LIN {X 0,Y 112.614,Z 722.748,A -85,B 0,C 180,E1 -26395.902,E2 -26395.902} C_VEL
LIN {X 0,Y 117.98,Z 722.724,A -85,B 0,C 180,E1 -26402.419,E2 -26402.419} C_VEL
LIN {X 0,Y 125.127,Z 721.325,A -85,B 0,C 180,E1 -26408.157,E2 -26408.157} C_VEL
LIN {X 0,Y 133.921,Z 718.463,A -85,B 0,C 180,E1 -26413.016,E2 -26413.016} C_VEL
LIN {X 0,Y 141.325,Z 715.337,A -85,B 0,C 180,E1 -26416.142,E2 -26416.142} C_VEL
LIN {X 0,Y 149.284,Z 711.254,A -85,B 0,C 180,E1 -26418.871,E2 -26418.871} C_VEL
LIN {X 0,Y 158.633,Z 705.602,A -85,B 0,C 180,E1 -26421.472,E2 -26421.472} C_VEL
LIN {X 0,Y 168.139,Z 698.779,A -85,B 0,C 180,E1 -26423.572,E2 -26423.572} C_VEL
LIN {X 0,Y 177.498,Z 690.89,A -85,B 0,C 180,E1 -26425.242,E2 -26425.242} C_VEL
LIN {X 0,Y 187.18,Z 681.241,A -85,B 0,C 180,E1 -26426.63,E2 -26426.63} C_VEL
LIN {X 0,Y 190.089,Z 677.932,A -85,B 0,C 180,E1 -26427.016,E2 -26427.016} C_VEL
LIN {X 0,Y 190.338,Z 677.404,A -85,B 0,C 180,E1 -26427.586,E2 -26427.586} C_VEL
LIN {X 0,Y 181.04,Z 686.04,A -85,B 0,C 180,E1 -26429.692,E2 -26429.692} C_VEL
LIN {X 0,Y 172.667,Z 692.227,A -85,B 0,C 180,E1 -26431.786,E2 -26431.786} C_VEL
LIN {X 0,Y 168.26,Z 695.049,A -85,B 0,C 180,E1 -26432.741,E2 -26432.741} C_VEL
LIN {X 0,Y 156.692,Z 701.204,A -85,B 0,C 180,E1 -26434.37,E2 -26434.37} C_VEL
LIN {X 0,Y 150.109,Z 703.856,A -85,B 0,C 180,E1 -26435.619,E2 -26435.619} C_VEL
LIN {X 0,Y 147.136,Z 704.728,A -85,B 0,C 180,E1 -26436.515,E2 -26436.515} C_VEL
LIN {X 0,Y 139.812,Z 706.451,A -85,B 0,C 180,E1 -26439.399,E2 -26439.399} C_VEL
LIN {X 0,Y 132.422,Z 707.283,A -85,B 0,C 180,E1 -26442.801,E2 -26442.801} C_VEL
LIN {X 0,Y 124.975,Z 707.111,A -85,B 0,C 180,E1 -26447.002,E2 -26447.002} C_VEL
LIN {X 0,Y 120.601,Z 706.402,A -85,B 0,C 180,E1 -26449.933,E2 -26449.933} C_VEL
LIN {X 0,Y 116.605,Z 705.225,A -85,B 0,C 180,E1 -26453.078,E2 -26453.078} C_VEL
LIN {X 0,Y 112.62,Z 703.398,A -85,B 0,C 180,E1 -26456.804,E2 -26456.804} C_VEL
LIN {X 0,Y 108.337,Z 700.237,A -85,B 0,C 180,E1 -26461.86,E2 -26461.86} C_VEL
LIN {X 0,Y 104.736,Z 695.693,A -85,B 0,C 180,E1 -26467.714,E2 -26467.714} C_VEL
LIN {X 0,Y 102.439,Z 690.321,A -85,B 0,C 180,E1 -26473.505,E2 -26473.505} C_VEL
LIN {X 0,Y 101.184,Z 683.981,A -85,B 0,C 180,E1 -26479.266,E2 -26479.266} C_VEL
LIN {X 0,Y 100.922,Z 675.313,A -85,B 0,C 180,E1 -26485.69,E2 -26485.69} C_VEL
LIN {X 0,Y 101.574,Z 666.056,A -85,B 0,C 180,E1 -26491.262,E2 -26491.262} C_VEL
LIN {X 0,Y 102.776,Z 655.496,A -85,B 0,C 180,E1 -26496.342,E2 -26496.342} C_VEL
LIN {X 0,Y 104.173,Z 644.669,A -85,B 0,C 180,E1 -26500.495,E2 -26500.495} C_VEL
LIN {X 0,Y 105.616,Z 633.785,A -85,B 0,C 180,E1 -26503.761,E2 -26503.761} C_VEL
LIN {X 0,Y 107.07,Z 621.558,A -85,B 0,C 180,E1 -26506.565,E2 -26506.565} C_VEL
LIN {X 0,Y 108.307,Z 608.423,A -85,B 0,C 180,E1 -26508.73,E2 -26508.73} C_VEL
LIN {X 0,Y 109.201,Z 592.336,A -85,B 0,C 180,E1 -26510.542,E2 -26510.542} C_VEL
LIN {X 0,Y 101.07,Z 563.812,A -85,B 0,C 180,E1 -26514.537,E2 -26514.537} C_VEL
LIN {X 0,Y 100.847,Z 562.869,A -85,B 0,C 180,E1 -26515.21,E2 -26515.21} C_VEL
LIN {X 0,Y 100.671,Z 562.758,A -85,B 0,C 180,E1 -26520.747,E2 -26520.747} C_VEL
LIN {X 0,Y 100.789,Z 562.741,A -85,B 0,C 180,E1 -26525.269,E2 -26525.269} C_VEL
LIN {X 0,Y 100.817,Z 562.74,A -85,B 0,C 180,E1 -26529.602,E2 -26529.602} C_VEL
LIN {X 0,Y 101.107,Z 562.702,A -85,B 0,C 180,E1 -26536.699,E2 -26536.699} C_VEL
LIN {X 0,Y 101.245,Z 562.678,A -85,B 0,C 180,E1 -26542.02,E2 -26542.02} C_VEL
LIN {X 0,Y 101.869,Z 562.602,A -85,B 0,C 180,E1 -26550,E2 -26550} C_VEL
LIN {X 0,Y 101.245,Z 562.683,A -85,B 0,C 180,E1 -26557.98,E2 -26557.98} C_VEL
LIN {X 0,Y 101.104,Z 562.702,A -85,B 0,C 180,E1 -26563.294,E2 -26563.294} C_VEL
LIN {X 0,Y 100.819,Z 562.733,A -85,B 0,C 180,E1 -26570.398,E2 -26570.398} C_VEL
LIN {X 0,Y 100.777,Z 562.743,A -85,B 0,C 180,E1 -26574.958,E2 -26574.958} C_VEL
LIN {X 0,Y 100.708,Z 562.752,A -85,B 0,C 180,E1 -26583.127,E2 -26583.127} C_VEL
LIN {X 0,Y 100.695,Z 562.753,A -85,B 0,C 180,E1 -26589.846,E2 -26589.846} C_VEL
LIN {X 0,Y 100.689,Z 562.747,A -85,B 0,C 180,E1 -26595.732,E2 -26595.732} C_VEL
LIN {X 0,Y 100.662,Z 562.758,A -85,B 0,C 180,E1 -26601.069,E2 -26601.069} C_VEL
LIN {X 0,Y 100.701,Z 562.751,A -85,B 0,C 180,E1 -26606.874,E2 -26606.874} C_VEL
LIN {X 0,Y 100.786,Z 562.739,A -85,B 0,C 180,E1 -26615.265,E2 -26615.265} C_VEL
LIN {X 0,Y 100.821,Z 562.738,A -85,B 0,C 180,E1 -26619.6,E2 -26619.6} C_VEL
LIN {X 0,Y 101.188,Z 562.693,A -85,B 0,C 180,E1 -26627.972,E2 -26627.972} C_VEL
LIN {X 0,Y 101.267,Z 562.675,A -85,B 0,C 180,E1 -26632.02,E2 -26632.02} C_VEL
LIN {X 0,Y 101.867,Z 562.601,A -85,B 0,C 180,E1 -26639.999,E2 -26639.999} C_VEL
LIN {X 0,Y 101.263,Z 562.678,A -85,B 0,C 180,E1 -26647.977,E2 -26647.977} C_VEL
LIN {X 0,Y 101.122,Z 562.701,A -85,B 0,C 180,E1 -26653.349,E2 -26653.349} C_VEL
LIN {X 0,Y 100.813,Z 562.736,A -85,B 0,C 180,E1 -26660.398,E2 -26660.398} C_VEL
LIN {X 0,Y 100.772,Z 562.741,A -85,B 0,C 180,E1 -26664.958,E2 -26664.958} C_VEL
LIN {X 0,Y 100.689,Z 562.753,A -85,B 0,C 180,E1 -26673.115,E2 -26673.115} C_VEL
LIN {X 0,Y 100.638,Z 562.761,A -85,B 0,C 180,E1 -26679.81,E2 -26679.81} C_VEL
LIN {X 0,Y 100.674,Z 562.757,A -85,B 0,C 180,E1 -26685.726,E2 -26685.726} C_VEL
LIN {X 0,Y 101.408,Z 562.905,A -85,B 0,C 180,E1 -26694.618,E2 -26694.618} C_VEL
LIN {X 0,Y 101.774,Z 563.975,A -85,B 0,C 180,E1 -26695.205,E2 -26695.205} C_VEL
LIN {X 0,Y 103.632,Z 569.648,A -85,B 0,C 180,E1 -26696.132,E2 -26696.132} C_VEL
LIN {X 0,Y 103.272,Z 600.843,A -85,B 0,C 180,E1 -26699.875,E2 -26699.875} C_VEL
LIN {X 0,Y 104.824,Z 644.068,A -85,B 0,C 180,E1 -26705.293,E2 -26705.293} C_VEL
LIN {X 0,Y 105.422,Z 656.065,A -85,B 0,C 180,E1 -26707.461,E2 -26707.461} C_VEL
LIN {X 0,Y 104.651,Z 667.818,A -85,B 0,C 180,E1 -26710.38,E2 -26710.38} C_VEL
LIN {X 0,Y 103.741,Z 677.783,A -85,B 0,C 180,E1 -26713.635,E2 -26713.635} C_VEL
LIN {X 0,Y 102.893,Z 688.58,A -85,B 0,C 180,E1 -26718.176,E2 -26718.176} C_VEL
LIN {X 0,Y 102.772,Z 696.112,A -85,B 0,C 180,E1 -26722.139,E2 -26722.139} C_VEL
LIN {X 0,Y 103.173,Z 703.754,A -85,B 0,C 180,E1 -26727.071,E2 -26727.071} C_VEL
LIN {X 0,Y 104.291,Z 709.858,A -85,B 0,C 180,E1 -26731.931,E2 -26731.931} C_VEL
LIN {X 0,Y 103.97,Z 711.518,A -85,B 0,C 180,E1 -26733.876,E2 -26733.876} C_VEL
LIN {X 0,Y 102.447,Z 715.261,A -85,B 0,C 180,E1 -26739.875,E2 -26739.875} C_VEL
LIN {X 0,Y 102.309,Z 718.051,A -85,B 0,C 180,E1 -26745.948,E2 -26745.948} C_VEL
LIN {X 0,Y 102.995,Z 719.41,A -85,B 0,C 180,E1 -26749.948,E2 -26749.948} C_VEL
LIN {X 0,Y 106.397,Z 721.105,A -85,B 0,C 180,E1 -26757.54,E2 -26757.54} C_VEL
LIN {X 0,Y 112.126,Z 721.458,A -85,B 0,C 180,E1 -26764.34,E2 -26764.34} C_VEL
LIN {X 0,Y 119.679,Z 720.429,A -85,B 0,C 180,E1 -26770.236,E2 -26770.236} C_VEL
LIN {X 0,Y 128.829,Z 718.027,A -85,B 0,C 180,E1 -26775.167,E2 -26775.167} C_VEL
LIN {X 0,Y 136.51,Z 715.246,A -85,B 0,C 180,E1 -26778.287,E2 -26778.287} C_VEL
LIN {X 0,Y 144.725,Z 711.612,A -85,B 0,C 180,E1 -26780.983,E2 -26780.983} C_VEL
LIN {X 0,Y 154.641,Z 706.256,A -85,B 0,C 180,E1 -26783.606,E2 -26783.606} C_VEL
LIN {X 0,Y 164.038,Z 700.248,A -85,B 0,C 180,E1 -26785.56,E2 -26785.56} C_VEL
LIN {X 0,Y 173.549,Z 693.028,A -85,B 0,C 180,E1 -26787.168,E2 -26787.168} C_VEL
LIN {X 0,Y 176.452,Z 690.599,A -85,B 0,C 180,E1 -26787.574,E2 -26787.574} C_VEL
LIN {X 0,Y 177.168,Z 689.792,A -85,B 0,C 180,E1 -26788.056,E2 -26788.056} C_VEL
LIN {X 0,Y 168.844,Z 695.339,A -85,B 0,C 180,E1 -26790.035,E2 -26790.035} C_VEL
LIN {X 0,Y 159.095,Z 700.398,A -85,B 0,C 180,E1 -26792.651,E2 -26792.651} C_VEL
LIN {X 0,Y 150.849,Z 703.626,A -85,B 0,C 180,E1 -26795.21,E2 -26795.21} C_VEL
LIN {X 0,Y 147.136,Z 704.728,A -85,B 0,C 180,E1 -26796.515,E2 -26796.515} C_VEL
LIN {X 0,Y 142.536,Z 706.017,A -85,B 0,C 180,E1 -26797.902,E2 -26797.902} C_VEL
LIN {X 0,Y 133.959,Z 707.764,A -85,B 0,C 180,E1 -26799.843,E2 -26799.843} C_VEL
LIN {X 0,Y 125.513,Z 708.563,A -85,B 0,C 180,E1 -26802.069,E2 -26802.069} C_VEL
LIN {X 0,Y 121.226,Z 708.373,A -85,B 0,C 180,E1 -26803.933,E2 -26803.933} C_VEL
LIN {X 0,Y 115.029,Z 707.323,A -85,B 0,C 180,E1 -26807.833,E2 -26807.833} C_VEL
LIN {X 0,Y 108.972,Z 705.197,A -85,B 0,C 180,E1 -26812.59,E2 -26812.59} C_VEL
LIN {X 0,Y 103.625,Z 701.961,A -85,B 0,C 180,E1 -26818.058,E2 -26818.058} C_VEL
LIN {X 0,Y 98.769,Z 696.798,A -85,B 0,C 180,E1 -26825.028,E2 -26825.028} C_VEL
LIN {X 0,Y 95.833,Z 690.877,A -85,B 0,C 180,E1 -26831.636,E2 -26831.636} C_VEL
LIN {X 0,Y 94.242,Z 683.557,A -85,B 0,C 180,E1 -26838.48,E2 -26838.48} C_VEL
LIN {X 0,Y 93.898,Z 674.309,A -85,B 0,C 180,E1 -26845.612,E2 -26845.612} C_VEL
LIN {X 0,Y 94.554,Z 664.987,A -85,B 0,C 180,E1 -26851.354,E2 -26851.354} C_VEL
LIN {X 0,Y 95.779,Z 654.409,A -85,B 0,C 180,E1 -26856.6,E2 -26856.6} C_VEL
LIN {X 0,Y 97.327,Z 642.456,A -85,B 0,C 180,E1 -26861.22,E2 -26861.22} C_VEL
LIN {X 0,Y 98.9,Z 630.748,A -85,B 0,C 180,E1 -26864.716,E2 -26864.716} C_VEL
LIN {X 0,Y 100.413,Z 617.425,A -85,B 0,C 180,E1 -26867.672,E2 -26867.672} C_VEL
LIN {X 0,Y 101.564,Z 603.656,A -85,B 0,C 180,E1 -26869.76,E2 -26869.76} C_VEL
LIN {X 0,Y 102.182,Z 593.607,A -85,B 0,C 180,E1 -26870.905,E2 -26870.905} C_VEL
LIN {X 0,Y 93.914,Z 564.332,A -85,B 0,C 180,E1 -26875.334,E2 -26875.334} C_VEL
LIN {X 0,Y 93.803,Z 563.659,A -85,B 0,C 180,E1 -26876.216,E2 -26876.216} C_VEL
LIN {X 0,Y 93.672,Z 563.629,A -85,B 0,C 180,E1 -26884.206,E2 -26884.206} C_VEL
LIN {X 0,Y 93.694,Z 563.627,A -85,B 0,C 180,E1 -26887.974,E2 -26887.974} C_VEL
LIN {X 0,Y 94.027,Z 563.584,A -85,B 0,C 180,E1 -26896.339,E2 -26896.339} C_VEL
LIN {X 0,Y 94.178,Z 563.559,A -85,B 0,C 180,E1 -26901.417,E2 -26901.417} C_VEL
LIN {X 0,Y 94.794,Z 563.483,A -85,B 0,C 180,E1 -26910,E2 -26910} C_VEL
LIN {X 0,Y 94.178,Z 563.562,A -85,B 0,C 180,E1 -26918.584,E2 -26918.584} C_VEL
LIN {X 0,Y 94.024,Z 563.585,A -85,B 0,C 180,E1 -26923.654,E2 -26923.654} C_VEL
LIN {X 0,Y 93.696,Z 563.625,A -85,B 0,C 180,E1 -26932.027,E2 -26932.027} C_VEL
LIN {X 0,Y 93.624,Z 563.63,A -85,B 0,C 180,E1 -26936.769,E2 -26936.769} C_VEL
LIN {X 0,Y 93.614,Z 563.634,A -85,B 0,C 180,E1 -26944.326,E2 -26944.326} C_VEL
LIN {X 0,Y 93.578,Z 563.64,A -85,B 0,C 180,E1 -26952.525,E2 -26952.525} C_VEL
LIN {X 0,Y 93.567,Z 563.642,A -85,B 0,C 180,E1 -26958.686,E2 -26958.686} C_VEL
LIN {X 0,Y 93.602,Z 563.631,A -85,B 0,C 180,E1 -26965.681,E2 -26965.681} C_VEL
LIN {X 0,Y 93.67,Z 563.621,A -85,B 0,C 180,E1 -26974.203,E2 -26974.203} C_VEL
LIN {X 0,Y 93.696,Z 563.626,A -85,B 0,C 180,E1 -26977.971,E2 -26977.971} C_VEL
LIN {X 0,Y 94.091,Z 563.577,A -85,B 0,C 180,E1 -26987.05,E2 -26987.05} C_VEL
LIN {X 0,Y 94.2,Z 563.554,A -85,B 0,C 180,E1 -26991.417,E2 -26991.417} C_VEL
LIN {X 0,Y 94.793,Z 563.482,A -85,B 0,C 180,E1 -26999.998,E2 -26999.998} C_VEL
LIN {X 0,Y 94.196,Z 563.556,A -85,B 0,C 180,E1 -27008.58,E2 -27008.58} C_VEL
LIN {X 0,Y 94.04,Z 563.583,A -85,B 0,C 180,E1 -27013.706,E2 -27013.706} C_VEL
LIN {X 0,Y 93.691,Z 563.626,A -85,B 0,C 180,E1 -27022.027,E2 -27022.027} C_VEL
LIN {X 0,Y 93.62,Z 563.627,A -85,B 0,C 180,E1 -27026.769,E2 -27026.769} C_VEL
LIN {X 0,Y 93.585,Z 563.635,A -85,B 0,C 180,E1 -27034.304,E2 -27034.304} C_VEL
LIN {X 0,Y 93.539,Z 563.644,A -85,B 0,C 180,E1 -27042.546,E2 -27042.546} C_VEL
LIN {X 0,Y 93.7,Z 563.626,A -85,B 0,C 180,E1 -27048.593,E2 -27048.593} C_VEL
LIN {X 0,Y 94.204,Z 563.779,A -85,B 0,C 180,E1 -27053.835,E2 -27053.835} C_VEL
LIN {X 0,Y 94.503,Z 564.713,A -85,B 0,C 180,E1 -27054.45,E2 -27054.45} C_VEL
LIN {X 0,Y 96.606,Z 570.603,A -85,B 0,C 180,E1 -27055.497,E2 -27055.497} C_VEL
LIN {X 0,Y 96.273,Z 602.738,A -85,B 0,C 180,E1 -27059.653,E2 -27059.653} C_VEL
LIN {X 0,Y 97.713,Z 642.777,A -85,B 0,C 180,E1 -27065.061,E2 -27065.061} C_VEL
LIN {X 0,Y 98.343,Z 655.818,A -85,B 0,C 180,E1 -27067.627,E2 -27067.627} C_VEL
LIN {X 0,Y 97.577,Z 667.437,A -85,B 0,C 180,E1 -27070.778,E2 -27070.778} C_VEL
LIN {X 0,Y 96.645,Z 678.326,A -85,B 0,C 180,E1 -27074.716,E2 -27074.716} C_VEL
LIN {X 0,Y 96.023,Z 687.428,A -85,B 0,C 180,E1 -27078.923,E2 -27078.923} C_VEL
LIN {X 0,Y 96.001,Z 695.694,A -85,B 0,C 180,E1 -27083.695,E2 -27083.695} C_VEL
LIN {X 0,Y 96.682,Z 703.137,A -85,B 0,C 180,E1 -27088.958,E2 -27088.958} C_VEL
LIN {X 0,Y 97.48,Z 706.871,A -85,B 0,C 180,E1 -27092.066,E2 -27092.066} C_VEL
LIN {X 0,Y 97.411,Z 708.801,A -85,B 0,C 180,E1 -27094.137,E2 -27094.137} C_VEL
LIN {X 0,Y 95.833,Z 712.817,A -85,B 0,C 180,E1 -27100.564,E2 -27100.564} C_VEL
LIN {X 0,Y 95.848,Z 716,A -85,B 0,C 180,E1 -27107.6,E2 -27107.6} C_VEL
LIN {X 0,Y 98.145,Z 718.518,A -85,B 0,C 180,E1 -27115.444,E2 -27115.444} C_VEL
LIN {X 0,Y 103.091,Z 719.881,A -85,B 0,C 180,E1 -27123.05,E2 -27123.05} C_VEL
LIN {X 0,Y 110.231,Z 719.92,A -85,B 0,C 180,E1 -27129.61,E2 -27129.61} C_VEL
LIN {X 0,Y 119.01,Z 718.623,A -85,B 0,C 180,E1 -27135.123,E2 -27135.123} C_VEL
LIN {X 0,Y 129.174,Z 715.958,A -85,B 0,C 180,E1 -27139.612,E2 -27139.612} C_VEL
LIN {X 0,Y 140.368,Z 711.805,A -85,B 0,C 180,E1 -27143.233,E2 -27143.233} C_VEL
LIN {X 0,Y 149.67,Z 707.434,A -85,B 0,C 180,E1 -27145.594,E2 -27145.594} C_VEL
LIN {X 0,Y 158.536,Z 702.476,A -85,B 0,C 180,E1 -27147.38,E2 -27147.38} C_VEL
LIN {X 0,Y 162.831,Z 699.761,A -85,B 0,C 180,E1 -27148.12,E2 -27148.12} C_VEL
LIN {X 0,Y 162.66,Z 699.588,A -85,B 0,C 180,E1 -27148.771,E2 -27148.771} C_VEL
LIN {X 0,Y 156.372,Z 702.462,A -85,B 0,C 180,E1 -27150.372,E2 -27150.372} C_VEL
LIN {X 0,Y 150.137,Z 704.754,A -85,B 0,C 180,E1 -27152.09,E2 -27152.09} C_VEL
LIN {X 0,Y 142.887,Z 706.741,A -85,B 0,C 180,E1 -27154.429,E2 -27154.429} C_VEL
LIN {X 0,Y 132.822,Z 708.424,A -85,B 0,C 180,E1 -27158.261,E2 -27158.261} C_VEL
LIN {X 0,Y 125.562,Z 708.674,A -85,B 0,C 180,E1 -27161.593,E2 -27161.593} C_VEL
LIN {X 0,Y 121.226,Z 708.373,A -85,B 0,C 180,E1 -27163.933,E2 -27163.933} C_VEL
LIN {X 0,Y 117.065,Z 707.982,A -85,B 0,C 180,E1 -27165.936,E2 -27165.936} C_VEL
LIN {X 0,Y 109.219,Z 706.798,A -85,B 0,C 180,E1 -27168.95,E2 -27168.95} C_VEL
LIN {X 0,Y 101.808,Z 704.734,A -85,B 0,C 180,E1 -27172.341,E2 -27172.341} C_VEL
LIN {X 0,Y 98.458,Z 702.962,A -85,B 0,C 180,E1 -27174.932,E2 -27174.932} C_VEL
LIN {X 0,Y 92.966,Z 697.676,A -85,B 0,C 180,E1 -27182.168,E2 -27182.168} C_VEL
LIN {X 0,Y 89.528,Z 691.801,A -85,B 0,C 180,E1 -27189.034,E2 -27189.034} C_VEL
LIN {X 0,Y 87.61,Z 685.1,A -85,B 0,C 180,E1 -27195.719,E2 -27195.719} C_VEL
LIN {X 0,Y 86.875,Z 676.928,A -85,B 0,C 180,E1 -27202.6,E2 -27202.6} C_VEL
LIN {X 0,Y 87.298,Z 666.901,A -85,B 0,C 180,E1 -27209.546,E2 -27209.546} C_VEL
LIN {X 0,Y 88.446,Z 655.795,A -85,B 0,C 180,E1 -27215.655,E2 -27215.655} C_VEL
LIN {X 0,Y 89.807,Z 645.151,A -85,B 0,C 180,E1 -27220.215,E2 -27220.215} C_VEL
LIN {X 0,Y 91.519,Z 632.797,A -85,B 0,C 180,E1 -27224.321,E2 -27224.321} C_VEL
LIN {X 0,Y 93.099,Z 619.497,A -85,B 0,C 180,E1 -27227.559,E2 -27227.559} C_VEL
LIN {X 0,Y 94.334,Z 606.24,A -85,B 0,C 180,E1 -27229.802,E2 -27229.802} C_VEL
LIN {X 0,Y 95.01,Z 594.162,A -85,B 0,C 180,E1 -27231.319,E2 -27231.319} C_VEL
LIN {X 0,Y 86.895,Z 565.312,A -85,B 0,C 180,E1 -27236.044,E2 -27236.044} C_VEL
LIN {X 0,Y 86.672,Z 564.554,A -85,B 0,C 180,E1 -27236.99,E2 -27236.99} C_VEL
LIN {X 0,Y 86.588,Z 564.511,A -85,B 0,C 180,E1 -27243.234,E2 -27243.234} C_VEL
LIN {X 0,Y 86.647,Z 564.502,A -85,B 0,C 180,E1 -27251.069,E2 -27251.069} C_VEL
LIN {X 0,Y 86.934,Z 564.466,A -85,B 0,C 180,E1 -27255.965,E2 -27255.965} C_VEL
LIN {X 0,Y 87.088,Z 564.445,A -85,B 0,C 180,E1 -27260.712,E2 -27260.712} C_VEL
LIN {X 0,Y 87.721,Z 564.364,A -85,B 0,C 180,E1 -27270,E2 -27270} C_VEL
LIN {X 0,Y 87.087,Z 564.442,A -85,B 0,C 180,E1 -27279.288,E2 -27279.288} C_VEL
LIN {X 0,Y 86.934,Z 564.469,A -85,B 0,C 180,E1 -27284.036,E2 -27284.036} C_VEL
LIN {X 0,Y 86.648,Z 564.495,A -85,B 0,C 180,E1 -27288.931,E2 -27288.931} C_VEL
LIN {X 0,Y 86.587,Z 564.506,A -85,B 0,C 180,E1 -27296.764,E2 -27296.764} C_VEL
LIN {X 0,Y 86.538,Z 564.511,A -85,B 0,C 180,E1 -27305.692,E2 -27305.692} C_VEL
LIN {X 0,Y 86.513,Z 564.519,A -85,B 0,C 180,E1 -27313.017,E2 -27313.017} C_VEL
LIN {X 0,Y 86.483,Z 564.524,A -85,B 0,C 180,E1 -27319.448,E2 -27319.448} C_VEL
LIN {X 0,Y 86.547,Z 564.508,A -85,B 0,C 180,E1 -27325.357,E2 -27325.357} C_VEL
LIN {X 0,Y 86.585,Z 564.503,A -85,B 0,C 180,E1 -27333.232,E2 -27333.232} C_VEL
LIN {X 0,Y 86.665,Z 564.497,A -85,B 0,C 180,E1 -27341.07,E2 -27341.07} C_VEL
LIN {X 0,Y 86.969,Z 564.463,A -85,B 0,C 180,E1 -27345.968,E2 -27345.968} C_VEL
LIN {X 0,Y 87.108,Z 564.438,A -85,B 0,C 180,E1 -27350.712,E2 -27350.712} C_VEL
LIN {X 0,Y 87.72,Z 564.362,A -85,B 0,C 180,E1 -27359.998,E2 -27359.998} C_VEL
LIN {X 0,Y 87.105,Z 564.438,A -85,B 0,C 180,E1 -27369.285,E2 -27369.285} C_VEL
LIN {X 0,Y 86.949,Z 564.467,A -85,B 0,C 180,E1 -27374.086,E2 -27374.086} C_VEL
LIN {X 0,Y 86.585,Z 564.511,A -85,B 0,C 180,E1 -27383.942,E2 -27383.942} C_VEL
LIN {X 0,Y 86.473,Z 564.522,A -85,B 0,C 180,E1 -27389.184,E2 -27389.184} C_VEL
LIN {X 0,Y 86.503,Z 564.513,A -85,B 0,C 180,E1 -27395.665,E2 -27395.665} C_VEL
LIN {X 0,Y 86.488,Z 564.522,A -85,B 0,C 180,E1 -27403.002,E2 -27403.002} C_VEL
LIN {X 0,Y 87.038,Z 564.64,A -85,B 0,C 180,E1 -27412.959,E2 -27412.959} C_VEL
LIN {X 0,Y 87.289,Z 565.429,A -85,B 0,C 180,E1 -27413.621,E2 -27413.621} C_VEL
LIN {X 0,Y 89.59,Z 572.071,A -85,B 0,C 180,E1 -27414.937,E2 -27414.937} C_VEL
LIN {X 0,Y 89.226,Z 603.646,A -85,B 0,C 180,E1 -27419.364,E2 -27419.364} C_VEL
LIN {X 0,Y 90.54,Z 641.544,A -85,B 0,C 180,E1 -27424.881,E2 -27424.881} C_VEL
LIN {X 0,Y 91.204,Z 654.519,A -85,B 0,C 180,E1 -27427.618,E2 -27427.618} C_VEL
LIN {X 0,Y 90.703,Z 664.594,A -85,B 0,C 180,E1 -27430.517,E2 -27430.517} C_VEL
LIN {X 0,Y 89.956,Z 674.381,A -85,B 0,C 180,E1 -27434.131,E2 -27434.131} C_VEL
LIN {X 0,Y 89.213,Z 684.978,A -85,B 0,C 180,E1 -27439.216,E2 -27439.216} C_VEL
LIN {X 0,Y 89.28,Z 693.53,A -85,B 0,C 180,E1 -27444.353,E2 -27444.353} C_VEL
LIN {X 0,Y 90.089,Z 701.136,A -85,B 0,C 180,E1 -27450,E2 -27450} C_VEL
LIN {X 0,Y 90.894,Z 704.957,A -85,B 0,C 180,E1 -27453.324,E2 -27453.324} C_VEL
LIN {X 0,Y 90.876,Z 705.941,A -85,B 0,C 180,E1 -27454.435,E2 -27454.435} C_VEL
LIN {X 0,Y 89.349,Z 710.165,A -85,B 0,C 180,E1 -27461.34,E2 -27461.34} C_VEL
LIN {X 0,Y 89.552,Z 713.951,A -85,B 0,C 180,E1 -27469.655,E2 -27469.655} C_VEL
LIN {X 0,Y 92.001,Z 716.468,A -85,B 0,C 180,E1 -27477.279,E2 -27477.279} C_VEL
LIN {X 0,Y 97.349,Z 718.193,A -85,B 0,C 180,E1 -27485.277,E2 -27485.277} C_VEL
LIN {X 0,Y 104.936,Z 718.599,A -85,B 0,C 180,E1 -27492.045,E2 -27492.045} C_VEL
LIN {X 0,Y 114.15,Z 717.73,A -85,B 0,C 180,E1 -27497.629,E2 -27497.629} C_VEL
LIN {X 0,Y 124.712,Z 715.5,A -85,B 0,C 180,E1 -27502.086,E2 -27502.086} C_VEL
LIN {X 0,Y 136.237,Z 711.881,A -85,B 0,C 180,E1 -27505.625,E2 -27505.625} C_VEL
LIN {X 0,Y 146.692,Z 707.546,A -85,B 0,C 180,E1 -27508.09,E2 -27508.09} C_VEL
LIN {X 0,Y 148.457,Z 706.694,A -85,B 0,C 180,E1 -27508.441,E2 -27508.441} C_VEL
LIN {X 0,Y 150.011,Z 705.845,A -85,B 0,C 180,E1 -27508.98,E2 -27508.98} C_VEL
LIN {X 0,Y 143.67,Z 707.653,A -85,B 0,C 180,E1 -27510.715,E2 -27510.715} C_VEL
LIN {X 0,Y 137.561,Z 708.931,A -85,B 0,C 180,E1 -27512.626,E2 -27512.626} C_VEL
LIN {X 0,Y 131.584,Z 709.723,A -85,B 0,C 180,E1 -27514.706,E2 -27514.706} C_VEL
LIN {X 0,Y 125.816,Z 710.066,A -85,B 0,C 180,E1 -27516.984,E2 -27516.984} C_VEL
LIN {X 0,Y 119.956,Z 709.899,A -85,B 0,C 180,E1 -27519.616,E2 -27519.616} C_VEL
LIN {X 0,Y 115.046,Z 709.332,A -85,B 0,C 180,E1 -27522.216,E2 -27522.216} C_VEL
LIN {X 0,Y 108.524,Z 707.824,A -85,B 0,C 180,E1 -27526.258,E2 -27526.258} C_VEL
LIN {X 0,Y 101.345,Z 704.812,A -85,B 0,C 180,E1 -27532.029,E2 -27532.029} C_VEL
LIN {X 0,Y 98.458,Z 702.962,A -85,B 0,C 180,E1 -27534.932,E2 -27534.932} C_VEL
LIN {X 0,Y 95.363,Z 700.961,A -85,B 0,C 180,E1 -27537.644,E2 -27537.644} C_VEL
LIN {X 0,Y 89.282,Z 697.082,A -85,B 0,C 180,E1 -27541.863,E2 -27541.863} C_VEL
LIN {X 0,Y 83.909,Z 692.396,A -85,B 0,C 180,E1 -27546.473,E2 -27546.473} C_VEL
LIN {X 0,Y 82.054,Z 689.238,A -85,B 0,C 180,E1 -27549.707,E2 -27549.707} C_VEL
LIN {X 0,Y 80.213,Z 680.7,A -85,B 0,C 180,E1 -27558.037,E2 -27558.037} C_VEL
LIN {X 0,Y 79.889,Z 672.496,A -85,B 0,C 180,E1 -27564.702,E2 -27564.702} C_VEL
LIN {X 0,Y 80.59,Z 662.201,A -85,B 0,C 180,E1 -27571.552,E2 -27571.552} C_VEL
LIN {X 0,Y 81.9,Z 651.041,A -85,B 0,C 180,E1 -27577.443,E2 -27577.443} C_VEL
LIN {X 0,Y 83.508,Z 639.148,A -85,B 0,C 180,E1 -27582.323,E2 -27582.323} C_VEL
LIN {X 0,Y 85.191,Z 626.492,A -85,B 0,C 180,E1 -27586.21,E2 -27586.21} C_VEL
LIN {X 0,Y 86.581,Z 613.937,A -85,B 0,C 180,E1 -27588.995,E2 -27588.995} C_VEL
LIN {X 0,Y 88.035,Z 595.646,A -85,B 0,C 180,E1 -27591.64,E2 -27591.64} C_VEL
LIN {X 0,Y 79.802,Z 566.307,A -85,B 0,C 180,E1 -27596.794,E2 -27596.794} C_VEL
LIN {X 0,Y 79.61,Z 565.44,A -85,B 0,C 180,E1 -27597.831,E2 -27597.831} C_VEL
LIN {X 0,Y 79.529,Z 565.392,A -85,B 0,C 180,E1 -27603.779,E2 -27603.779} C_VEL
LIN {X 0,Y 79.515,Z 565.393,A -85,B 0,C 180,E1 -27609.297,E2 -27609.297} C_VEL
LIN {X 0,Y 79.828,Z 565.349,A -85,B 0,C 180,E1 -27615.574,E2 -27615.574} C_VEL
LIN {X 0,Y 79.971,Z 565.333,A -85,B 0,C 180,E1 -27619.877,E2 -27619.877} C_VEL
LIN {X 0,Y 80.648,Z 565.245,A -85,B 0,C 180,E1 -27630,E2 -27630} C_VEL
LIN {X 0,Y 79.97,Z 565.327,A -85,B 0,C 180,E1 -27640.123,E2 -27640.123} C_VEL
LIN {X 0,Y 79.747,Z 565.364,A -85,B 0,C 180,E1 -27645.33,E2 -27645.33} C_VEL
LIN {X 0,Y 79.516,Z 565.387,A -85,B 0,C 180,E1 -27650.704,E2 -27650.704} C_VEL
LIN {X 0,Y 79.485,Z 565.387,A -85,B 0,C 180,E1 -27657.844,E2 -27657.844} C_VEL
LIN {X 0,Y 79.395,Z 565.408,A -85,B 0,C 180,E1 -27662.08,E2 -27662.08} C_VEL
LIN {X 0,Y 79.395,Z 565.4,A -85,B 0,C 180,E1 -27668.289,E2 -27668.289} C_VEL
LIN {X 0,Y 79.419,Z 565.397,A -85,B 0,C 180,E1 -27675.067,E2 -27675.067} C_VEL
LIN {X 0,Y 79.401,Z 565.403,A -85,B 0,C 180,E1 -27682.807,E2 -27682.807} C_VEL
LIN {X 0,Y 79.387,Z 565.407,A -85,B 0,C 180,E1 -27687.913,E2 -27687.913} C_VEL
LIN {X 0,Y 79.526,Z 565.382,A -85,B 0,C 180,E1 -27693.775,E2 -27693.775} C_VEL
LIN {X 0,Y 79.524,Z 565.391,A -85,B 0,C 180,E1 -27699.296,E2 -27699.296} C_VEL
LIN {X 0,Y 79.842,Z 565.351,A -85,B 0,C 180,E1 -27705.523,E2 -27705.523} C_VEL
LIN {X 0,Y 79.993,Z 565.327,A -85,B 0,C 180,E1 -27709.878,E2 -27709.878} C_VEL
LIN {X 0,Y 80.648,Z 565.243,A -85,B 0,C 180,E1 -27719.998,E2 -27719.998} C_VEL
LIN {X 0,Y 79.99,Z 565.325,A -85,B 0,C 180,E1 -27730.119,E2 -27730.119} C_VEL
LIN {X 0,Y 79.761,Z 565.36,A -85,B 0,C 180,E1 -27735.326,E2 -27735.326} C_VEL
LIN {X 0,Y 79.511,Z 565.39,A -85,B 0,C 180,E1 -27740.703,E2 -27740.703} C_VEL
LIN {X 0,Y 79.48,Z 565.389,A -85,B 0,C 180,E1 -27747.842,E2 -27747.842} C_VEL
LIN {X 0,Y 79.375,Z 565.41,A -85,B 0,C 180,E1 -27752.088,E2 -27752.088} C_VEL
LIN {X 0,Y 79.364,Z 565.408,A -85,B 0,C 180,E1 -27758.305,E2 -27758.305} C_VEL
LIN {X 0,Y 79.442,Z 565.403,A -85,B 0,C 180,E1 -27765.049,E2 -27765.049} C_VEL
LIN {X 0,Y 79.912,Z 565.6,A -85,B 0,C 180,E1 -27772.213,E2 -27772.213} C_VEL
LIN {X 0,Y 80.171,Z 566.484,A -85,B 0,C 180,E1 -27772.859,E2 -27772.859} C_VEL
LIN {X 0,Y 82.536,Z 573.093,A -85,B 0,C 180,E1 -27774.248,E2 -27774.248} C_VEL
LIN {X 0,Y 82.268,Z 609.726,A -85,B 0,C 180,E1 -27779.875,E2 -27779.875} C_VEL
LIN {X 0,Y 83.447,Z 640.405,A -85,B 0,C 180,E1 -27784.763,E2 -27784.763} C_VEL
LIN {X 0,Y 84.032,Z 652.558,A -85,B 0,C 180,E1 -27787.516,E2 -27787.516} C_VEL
LIN {X 0,Y 83.971,Z 659.247,A -85,B 0,C 180,E1 -27789.464,E2 -27789.464} C_VEL
LIN {X 0,Y 83.298,Z 670.161,A -85,B 0,C 180,E1 -27793.456,E2 -27793.456} C_VEL
LIN {X 0,Y 82.526,Z 680.316,A -85,B 0,C 180,E1 -27798.331,E2 -27798.331} C_VEL
LIN {X 0,Y 82.516,Z 689.541,A -85,B 0,C 180,E1 -27803.888,E2 -27803.888} C_VEL
LIN {X 0,Y 83.287,Z 697.673,A -85,B 0,C 180,E1 -27810,E2 -27810} C_VEL
LIN {X 0,Y 84.42,Z 702.905,A -85,B 0,C 180,E1 -27814.775,E2 -27814.775} C_VEL
LIN {X 0,Y 82.914,Z 707.425,A -85,B 0,C 180,E1 -27822.234,E2 -27822.234} C_VEL
LIN {X 0,Y 83.02,Z 710.914,A -85,B 0,C 180,E1 -27829.792,E2 -27829.792} C_VEL
LIN {X 0,Y 85.997,Z 714.314,A -85,B 0,C 180,E1 -27839.362,E2 -27839.362} C_VEL
LIN {X 0,Y 91.822,Z 716.359,A -85,B 0,C 180,E1 -27847.756,E2 -27847.756} C_VEL
LIN {X 0,Y 99.865,Z 717.171,A -85,B 0,C 180,E1 -27854.727,E2 -27854.727} C_VEL
LIN {X 0,Y 109.535,Z 716.682,A -85,B 0,C 180,E1 -27860.347,E2 -27860.347} C_VEL
LIN {X 0,Y 120.505,Z 714.906,A -85,B 0,C 180,E1 -27864.733,E2 -27864.733} C_VEL
LIN {X 0,Y 132.363,Z 711.807,A -85,B 0,C 180,E1 -27868.159,E2 -27868.159} C_VEL
LIN {X 0,Y 135.122,Z 710.886,A -85,B 0,C 180,E1 -27868.813,E2 -27868.813} C_VEL
LIN {X 0,Y 136.15,Z 710.367,A -85,B 0,C 180,E1 -27869.503,E2 -27869.503} C_VEL
LIN {X 0,Y 124.78,Z 711.419,A -85,B 0,C 180,E1 -27873.22,E2 -27873.22} C_VEL
LIN {X 0,Y 115.71,Z 711.047,A -85,B 0,C 180,E1 -27876.892,E2 -27876.892} C_VEL
LIN {X 0,Y 107.749,Z 709.787,A -85,B 0,C 180,E1 -27880.967,E2 -27880.967} C_VEL
LIN {X 0,Y 102.104,Z 708.1,A -85,B 0,C 180,E1 -27884.497,E2 -27884.497} C_VEL
LIN {X 0,Y 95.808,Z 705.236,A -85,B 0,C 180,E1 -27889.434,E2 -27889.434} C_VEL
LIN {X 0,Y 89.905,Z 701.096,A -85,B 0,C 180,E1 -27895.518,E2 -27895.518} C_VEL
LIN {X 0,Y 85.562,Z 696.165,A -85,B 0,C 180,E1 -27901.878,E2 -27901.878} C_VEL
LIN {X 0,Y 82.054,Z 689.238,A -85,B 0,C 180,E1 -27909.707,E2 -27909.707} C_VEL
LIN {X 0,Y 80.513,Z 685.919,A -85,B 0,C 180,E1 -27912.939,E2 -27912.939} C_VEL
LIN {X 0,Y 76.802,Z 679.791,A -85,B 0,C 180,E1 -27917.907,E2 -27917.907} C_VEL
LIN {X 0,Y 73.624,Z 672.989,A -85,B 0,C 180,E1 -27922.954,E2 -27922.954} C_VEL
LIN {X 0,Y 73.02,Z 668.647,A -85,B 0,C 180,E1 -27926.142,E2 -27926.142} C_VEL
LIN {X 0,Y 73.795,Z 658.917,A -85,B 0,C 180,E1 -27932.659,E2 -27932.659} C_VEL
LIN {X 0,Y 75.116,Z 648.27,A -85,B 0,C 180,E1 -27938.307,E2 -27938.307} C_VEL
LIN {X 0,Y 76.825,Z 635.781,A -85,B 0,C 180,E1 -27943.417,E2 -27943.417} C_VEL
LIN {X 0,Y 78.468,Z 623.339,A -85,B 0,C 180,E1 -27947.168,E2 -27947.168} C_VEL
LIN {X 0,Y 79.828,Z 610.28,A -85,B 0,C 180,E1 -27949.967,E2 -27949.967} C_VEL
LIN {X 0,Y 80.842,Z 596.222,A -85,B 0,C 180,E1 -27952.092,E2 -27952.092} C_VEL
LIN {X 0,Y 72.7,Z 567.049,A -85,B 0,C 180,E1 -27957.759,E2 -27957.759} C_VEL
LIN {X 0,Y 72.495,Z 566.324,A -85,B 0,C 180,E1 -27958.841,E2 -27958.841} C_VEL
LIN {X 0,Y 72.396,Z 566.277,A -85,B 0,C 180,E1 -27967.152,E2 -27967.152} C_VEL
LIN {X 0,Y 72.724,Z 566.233,A -85,B 0,C 180,E1 -27975.111,E2 -27975.111} C_VEL
LIN {X 0,Y 72.862,Z 566.221,A -85,B 0,C 180,E1 -27978.878,E2 -27978.878} C_VEL
LIN {X 0,Y 73.574,Z 566.126,A -85,B 0,C 180,E1 -27990,E2 -27990} C_VEL
LIN {X 0,Y 72.861,Z 566.213,A -85,B 0,C 180,E1 -28001.123,E2 -28001.123} C_VEL
LIN {X 0,Y 72.577,Z 566.254,A -85,B 0,C 180,E1 -28006.888,E2 -28006.888} C_VEL
LIN {X 0,Y 72.397,Z 566.279,A -85,B 0,C 180,E1 -28012.849,E2 -28012.849} C_VEL
LIN {X 0,Y 72.379,Z 566.274,A -85,B 0,C 180,E1 -28019.081,E2 -28019.081} C_VEL
LIN {X 0,Y 72.315,Z 566.282,A -85,B 0,C 180,E1 -28025.669,E2 -28025.669} C_VEL
LIN {X 0,Y 72.273,Z 566.293,A -85,B 0,C 180,E1 -28032.898,E2 -28032.898} C_VEL
LIN {X 0,Y 72.309,Z 566.29,A -85,B 0,C 180,E1 -28041.036,E2 -28041.036} C_VEL
LIN {X 0,Y 72.305,Z 566.281,A -85,B 0,C 180,E1 -28044.322,E2 -28044.322} C_VEL
LIN {X 0,Y 72.393,Z 566.278,A -85,B 0,C 180,E1 -28050.959,E2 -28050.959} C_VEL
LIN {X 0,Y 72.4,Z 566.279,A -85,B 0,C 180,E1 -28057.15,E2 -28057.15} C_VEL
LIN {X 0,Y 72.757,Z 566.231,A -85,B 0,C 180,E1 -28065.002,E2 -28065.002} C_VEL
LIN {X 0,Y 72.88,Z 566.217,A -85,B 0,C 180,E1 -28068.878,E2 -28068.878} C_VEL
LIN {X 0,Y 73.575,Z 566.124,A -85,B 0,C 180,E1 -28079.998,E2 -28079.998} C_VEL
LIN {X 0,Y 72.878,Z 566.214,A -85,B 0,C 180,E1 -28091.118,E2 -28091.118} C_VEL
LIN {X 0,Y 72.581,Z 566.249,A -85,B 0,C 180,E1 -28096.885,E2 -28096.885} C_VEL
LIN {X 0,Y 72.392,Z 566.28,A -85,B 0,C 180,E1 -28102.849,E2 -28102.849} C_VEL
LIN {X 0,Y 72.375,Z 566.277,A -85,B 0,C 180,E1 -28109.081,E2 -28109.081} C_VEL
LIN {X 0,Y 72.292,Z 566.283,A -85,B 0,C 180,E1 -28115.681,E2 -28115.681} C_VEL
LIN {X 0,Y 72.276,Z 566.292,A -85,B 0,C 180,E1 -28122.893,E2 -28122.893} C_VEL
LIN {X 0,Y 72.747,Z 566.465,A -85,B 0,C 180,E1 -28131.199,E2 -28131.199} C_VEL
LIN {X 0,Y 73.112,Z 567.625,A -85,B 0,C 180,E1 -28132.032,E2 -28132.032} C_VEL
LIN {X 0,Y 75.398,Z 574.035,A -85,B 0,C 180,E1 -28133.498,E2 -28133.498} C_VEL
LIN {X 0,Y 75.415,Z 620.491,A -85,B 0,C 180,E1 -28141.306,E2 -28141.306} C_VEL
LIN {X 0,Y 76.364,Z 640.892,A -85,B 0,C 180,E1 -28144.968,E2 -28144.968} C_VEL
LIN {X 0,Y 77.067,Z 654.644,A -85,B 0,C 180,E1 -28148.607,E2 -28148.607} C_VEL
LIN {X 0,Y 76.567,Z 665.625,A -85,B 0,C 180,E1 -28152.644,E2 -28152.644} C_VEL
LIN {X 0,Y 75.921,Z 675.277,A -85,B 0,C 180,E1 -28157.299,E2 -28157.299} C_VEL
LIN {X 0,Y 75.777,Z 685.167,A -85,B 0,C 180,E1 -28163.342,E2 -28163.342} C_VEL
LIN {X 0,Y 76.503,Z 693.909,A -85,B 0,C 180,E1 -28170,E2 -28170} C_VEL
LIN {X 0,Y 77.748,Z 699.588,A -85,B 0,C 180,E1 -28175.186,E2 -28175.186} C_VEL
LIN {X 0,Y 77.773,Z 700.511,A -85,B 0,C 180,E1 -28176.282,E2 -28176.282} C_VEL
LIN {X 0,Y 76.443,Z 705.895,A -85,B 0,C 180,E1 -28186.01,E2 -28186.01} C_VEL
LIN {X 0,Y 78.093,Z 710.324,A -85,B 0,C 180,E1 -28196.741,E2 -28196.741} C_VEL
LIN {X 0,Y 83.023,Z 713.359,A -85,B 0,C 180,E1 -28206.337,E2 -28206.337} C_VEL
LIN {X 0,Y 90.542,Z 715.177,A -85,B 0,C 180,E1 -28214.313,E2 -28214.313} C_VEL
LIN {X 0,Y 99.952,Z 715.694,A -85,B 0,C 180,E1 -28220.663,E2 -28220.663} C_VEL
LIN {X 0,Y 110.758,Z 714.997,A -85,B 0,C 180,E1 -28225.575,E2 -28225.575} C_VEL
LIN {X 0,Y 122.59,Z 713.053,A -85,B 0,C 180,E1 -28229.307,E2 -28229.307} C_VEL
LIN {X 0,Y 121.225,Z 712.804,A -85,B 0,C 180,E1 -28230.412,E2 -28230.412} C_VEL
LIN {X 0,Y 111.092,Z 712.101,A -85,B 0,C 180,E1 -28234.225,E2 -28234.225} C_VEL
LIN {X 0,Y 106.023,Z 711.257,A -85,B 0,C 180,E1 -28236.565,E2 -28236.565} C_VEL
LIN {X 0,Y 95.82,Z 708.17,A -85,B 0,C 180,E1 -28242.453,E2 -28242.453} C_VEL
LIN {X 0,Y 88.205,Z 704.239,A -85,B 0,C 180,E1 -28248.512,E2 -28248.512} C_VEL
LIN {X 0,Y 82.231,Z 699.411,A -85,B 0,C 180,E1 -28255.099,E2 -28255.099} C_VEL
LIN {X 0,Y 77.413,Z 693.012,A -85,B 0,C 180,E1 -28263.012,E2 -28263.012} C_VEL
LIN {X 0,Y 74.558,Z 685.892,A -85,B 0,C 180,E1 -28270.869,E2 -28270.869} C_VEL
LIN {X 0,Y 73.18,Z 678.338,A -85,B 0,C 180,E1 -28278.189,E2 -28278.189} C_VEL
LIN {X 0,Y 73.02,Z 668.647,A -85,B 0,C 180,E1 -28286.142,E2 -28286.142} C_VEL
LIN {X 0,Y 72.607,Z 664.26,A -85,B 0,C 180,E1 -28289.149,E2 -28289.149} C_VEL
LIN {X 0,Y 70.514,Z 656.427,A -85,B 0,C 180,E1 -28293.655,E2 -28293.655} C_VEL
LIN {X 0,Y 68.656,Z 648.054,A -85,B 0,C 180,E1 -28297.937,E2 -28297.937} C_VEL
LIN {X 0,Y 68.69,Z 642.762,A -85,B 0,C 180,E1 -28300.415,E2 -28300.415} C_VEL
LIN {X 0,Y 70.285,Z 631.381,A -85,B 0,C 180,E1 -28304.911,E2 -28304.911} C_VEL
LIN {X 0,Y 72.007,Z 617.616,A -85,B 0,C 180,E1 -28308.805,E2 -28308.805} C_VEL
LIN {X 0,Y 73.459,Z 601.642,A -85,B 0,C 180,E1 -28311.747,E2 -28311.747} C_VEL
LIN {X 0,Y 73.666,Z 596.873,A -85,B 0,C 180,E1 -28312.521,E2 -28312.521} C_VEL
LIN {X 0,Y 65.717,Z 568.366,A -85,B 0,C 180,E1 -28318.589,E2 -28318.589} C_VEL
LIN {X 0,Y 65.452,Z 567.294,A -85,B 0,C 180,E1 -28319.63,E2 -28319.63} C_VEL
LIN {X 0,Y 65.383,Z 567.149,A -85,B 0,C 180,E1 -28331.189,E2 -28331.189} C_VEL
LIN {X 0,Y 65.758,Z 567.107,A -85,B 0,C 180,E1 -28337.658,E2 -28337.658} C_VEL
LIN {X 0,Y 66.497,Z 567.007,A -85,B 0,C 180,E1 -28350,E2 -28350} C_VEL
LIN {X 0,Y 65.758,Z 567.101,A -85,B 0,C 180,E1 -28362.343,E2 -28362.343} C_VEL
LIN {X 0,Y 65.382,Z 567.143,A -85,B 0,C 180,E1 -28368.813,E2 -28368.813} C_VEL
LIN {X 0,Y 65.249,Z 567.167,A -85,B 0,C 180,E1 -28375.521,E2 -28375.521} C_VEL
LIN {X 0,Y 65.206,Z 567.175,A -85,B 0,C 180,E1 -28382.609,E2 -28382.609} C_VEL
LIN {X 0,Y 65.208,Z 567.175,A -85,B 0,C 180,E1 -28391.02,E2 -28391.02} C_VEL
LIN {X 0,Y 65.22,Z 567.173,A -85,B 0,C 180,E1 -28399.715,E2 -28399.715} C_VEL
LIN {X 0,Y 65.256,Z 567.169,A -85,B 0,C 180,E1 -28409.494,E2 -28409.494} C_VEL
LIN {X 0,Y 65.249,Z 567.161,A -85,B 0,C 180,E1 -28414.477,E2 -28414.477} C_VEL
LIN {X 0,Y 65.652,Z 567.114,A -85,B 0,C 180,E1 -28424.458,E2 -28424.458} C_VEL
LIN {X 0,Y 65.78,Z 567.104,A -85,B 0,C 180,E1 -28427.66,E2 -28427.66} C_VEL
LIN {X 0,Y 66.499,Z 567.005,A -85,B 0,C 180,E1 -28439.998,E2 -28439.998} C_VEL
LIN {X 0,Y 65.771,Z 567.103,A -85,B 0,C 180,E1 -28452.338,E2 -28452.338} C_VEL
LIN {X 0,Y 65.383,Z 567.144,A -85,B 0,C 180,E1 -28458.81,E2 -28458.81} C_VEL
LIN {X 0,Y 65.236,Z 567.164,A -85,B 0,C 180,E1 -28465.524,E2 -28465.524} C_VEL
LIN {X 0,Y 65.193,Z 567.176,A -85,B 0,C 180,E1 -28472.614,E2 -28472.614} C_VEL
LIN {X 0,Y 65.199,Z 567.176,A -85,B 0,C 180,E1 -28481.015,E2 -28481.015} C_VEL
LIN {X 0,Y 65.582,Z 567.315,A -85,B 0,C 180,E1 -28489.986,E2 -28489.986} C_VEL
LIN {X 0,Y 65.913,Z 568.396,A -85,B 0,C 180,E1 -28490.979,E2 -28490.979} C_VEL
LIN {X 0,Y 68.413,Z 576.041,A -85,B 0,C 180,E1 -28492.903,E2 -28492.903} C_VEL
LIN {X 0,Y 68.28,Z 618.926,A -85,B 0,C 180,E1 -28500.9,E2 -28500.9} C_VEL
LIN {X 0,Y 69.228,Z 640.077,A -85,B 0,C 180,E1 -28505.104,E2 -28505.104} C_VEL
LIN {X 0,Y 70.009,Z 653.57,A -85,B 0,C 180,E1 -28509.045,E2 -28509.045} C_VEL
LIN {X 0,Y 69.668,Z 663.754,A -85,B 0,C 180,E1 -28513.141,E2 -28513.141} C_VEL
LIN {X 0,Y 69.152,Z 673.563,A -85,B 0,C 180,E1 -28518.272,E2 -28518.272} C_VEL
LIN {X 0,Y 69.079,Z 682.556,A -85,B 0,C 180,E1 -28524.16,E2 -28524.16} C_VEL
LIN {X 0,Y 69.72,Z 689.925,A -85,B 0,C 180,E1 -28530,E2 -28530} C_VEL
LIN {X 0,Y 71.368,Z 697.208,A -85,B 0,C 180,E1 -28536.848,E2 -28536.848} C_VEL
LIN {X 0,Y 70.303,Z 701.504,A -85,B 0,C 180,E1 -28544.472,E2 -28544.472} C_VEL
LIN {X 0,Y 71.214,Z 706.401,A -85,B 0,C 180,E1 -28555.637,E2 -28555.637} C_VEL
LIN {X 0,Y 74.576,Z 709.548,A -85,B 0,C 180,E1 -28564.431,E2 -28564.431} C_VEL
LIN {X 0,Y 81.442,Z 712.354,A -85,B 0,C 180,E1 -28573.657,E2 -28573.657} C_VEL
LIN {X 0,Y 90.544,Z 713.86,A -85,B 0,C 180,E1 -28580.912,E2 -28580.912} C_VEL
LIN {X 0,Y 101.198,Z 714.183,A -85,B 0,C 180,E1 -28586.445,E2 -28586.445} C_VEL
LIN {X 0,Y 106.956,Z 713.899,A -85,B 0,C 180,E1 -28588.671,E2 -28588.671} C_VEL
LIN {X 0,Y 109.231,Z 713.411,A -85,B 0,C 180,E1 -28590.368,E2 -28590.368} C_VEL
LIN {X 0,Y 98.969,Z 711.319,A -85,B 0,C 180,E1 -28594.783,E2 -28594.783} C_VEL
LIN {X 0,Y 89.676,Z 707.98,A -85,B 0,C 180,E1 -28600.123,E2 -28600.123} C_VEL
LIN {X 0,Y 80.772,Z 702.867,A -85,B 0,C 180,E1 -28607.372,E2 -28607.372} C_VEL
LIN {X 0,Y 73.787,Z 696.218,A -85,B 0,C 180,E1 -28615.905,E2 -28615.905} C_VEL
LIN {X 0,Y 69.684,Z 689.757,A -85,B 0,C 180,E1 -28623.667,E2 -28623.667} C_VEL
LIN {X 0,Y 66.873,Z 680.811,A -85,B 0,C 180,E1 -28633.408,E2 -28633.408} C_VEL
LIN {X 0,Y 66.034,Z 670.757,A -85,B 0,C 180,E1 -28642.696,E2 -28642.696} C_VEL
LIN {X 0,Y 66.66,Z 659.834,A -85,B 0,C 180,E1 -28650.931,E2 -28650.931} C_VEL
LIN {X 0,Y 67.9,Z 648.812,A -85,B 0,C 180,E1 -28657.461,E2 -28657.461} C_VEL
LIN {X 0,Y 68.69,Z 642.762,A -85,B 0,C 180,E1 -28660.415,E2 -28660.415} C_VEL
LIN {X 0,Y 68.745,Z 637.533,A -85,B 0,C 180,E1 -28662.632,E2 -28662.632} C_VEL
LIN {X 0,Y 67.103,Z 628.585,A -85,B 0,C 180,E1 -28665.827,E2 -28665.827} C_VEL
LIN {X 0,Y 65.402,Z 619.222,A -85,B 0,C 180,E1 -28668.618,E2 -28668.618} C_VEL
LIN {X 0,Y 65.335,Z 613.431,A -85,B 0,C 180,E1 -28670.043,E2 -28670.043} C_VEL
LIN {X 0,Y 66.571,Z 597.736,A -85,B 0,C 180,E1 -28672.982,E2 -28672.982} C_VEL
LIN {X 0,Y 58.552,Z 568.995,A -85,B 0,C 180,E1 -28679.795,E2 -28679.795} C_VEL
LIN {X 0,Y 58.325,Z 568.103,A -85,B 0,C 180,E1 -28681.186,E2 -28681.186} C_VEL
LIN {X 0,Y 58.52,Z 567.998,A -85,B 0,C 180,E1 -28693.908,E2 -28693.908} C_VEL
LIN {X 0,Y 58.802,Z 567.963,A -85,B 0,C 180,E1 -28703.136,E2 -28703.136} C_VEL
LIN {X 0,Y 59.387,Z 567.892,A -85,B 0,C 180,E1 -28710,E2 -28710} C_VEL
LIN {X 0,Y 58.802,Z 567.972,A -85,B 0,C 180,E1 -28716.865,E2 -28716.865} C_VEL
LIN {X 0,Y 58.52,Z 568.006,A -85,B 0,C 180,E1 -28726.093,E2 -28726.093} C_VEL
LIN {X 0,Y 58.156,Z 568.044,A -85,B 0,C 180,E1 -28738.907,E2 -28738.907} C_VEL
LIN {X 0,Y 58.049,Z 568.056,A -85,B 0,C 180,E1 -28747.254,E2 -28747.254} C_VEL
LIN {X 0,Y 58.031,Z 568.059,A -85,B 0,C 180,E1 -28756.605,E2 -28756.605} C_VEL
LIN {X 0,Y 58.043,Z 568.062,A -85,B 0,C 180,E1 -28762.738,E2 -28762.738} C_VEL
LIN {X 0,Y 58.155,Z 568.05,A -85,B 0,C 180,E1 -28771.09,E2 -28771.09} C_VEL
LIN {X 0,Y 58.538,Z 567.998,A -85,B 0,C 180,E1 -28783.834,E2 -28783.834} C_VEL
LIN {X 0,Y 58.818,Z 567.964,A -85,B 0,C 180,E1 -28793.135,E2 -28793.135} C_VEL
LIN {X 0,Y 59.39,Z 567.89,A -85,B 0,C 180,E1 -28799.998,E2 -28799.998} C_VEL
LIN {X 0,Y 58.814,Z 567.967,A -85,B 0,C 180,E1 -28806.861,E2 -28806.861} C_VEL
LIN {X 0,Y 58.524,Z 568.002,A -85,B 0,C 180,E1 -28816.12,E2 -28816.12} C_VEL
LIN {X 0,Y 58.148,Z 568.048,A -85,B 0,C 180,E1 -28828.909,E2 -28828.909} C_VEL
LIN {X 0,Y 58.038,Z 568.06,A -85,B 0,C 180,E1 -28837.26,E2 -28837.26} C_VEL
LIN {X 0,Y 58.46,Z 568.258,A -85,B 0,C 180,E1 -28848.869,E2 -28848.869} C_VEL
LIN {X 0,Y 58.71,Z 569.039,A -85,B 0,C 180,E1 -28849.738,E2 -28849.738} C_VEL
LIN {X 0,Y 61.359,Z 577.539,A -85,B 0,C 180,E1 -28852.122,E2 -28852.122} C_VEL
LIN {X 0,Y 61.23,Z 620.961,A -85,B 0,C 180,E1 -28861.156,E2 -28861.156} C_VEL
LIN {X 0,Y 62.097,Z 639.36,A -85,B 0,C 180,E1 -28865.309,E2 -28865.309} C_VEL
LIN {X 0,Y 62.921,Z 652.434,A -85,B 0,C 180,E1 -28869.588,E2 -28869.588} C_VEL
LIN {X 0,Y 62.841,Z 660.168,A -85,B 0,C 180,E1 -28872.928,E2 -28872.928} C_VEL
LIN {X 0,Y 62.499,Z 669.27,A -85,B 0,C 180,E1 -28877.828,E2 -28877.828} C_VEL
LIN {X 0,Y 62.435,Z 679.847,A -85,B 0,C 180,E1 -28885.157,E2 -28885.157} C_VEL
LIN {X 0,Y 63.277,Z 687.495,A -85,B 0,C 180,E1 -28891.672,E2 -28891.672} C_VEL
LIN {X 0,Y 64.751,Z 693.564,A -85,B 0,C 180,E1 -28897.673,E2 -28897.673} C_VEL
LIN {X 0,Y 64.941,Z 695.026,A -85,B 0,C 180,E1 -28899.503,E2 -28899.503} C_VEL
LIN {X 0,Y 64.371,Z 701.279,A -85,B 0,C 180,E1 -28912.464,E2 -28912.464} C_VEL
LIN {X 0,Y 67.053,Z 705.375,A -85,B 0,C 180,E1 -28923.021,E2 -28923.021} C_VEL
LIN {X 0,Y 72.618,Z 708.716,A -85,B 0,C 180,E1 -28932.644,E2 -28932.644} C_VEL
LIN {X 0,Y 81.329,Z 711.202,A -85,B 0,C 180,E1 -28941.051,E2 -28941.051} C_VEL
LIN {X 0,Y 91.795,Z 712.495,A -85,B 0,C 180,E1 -28947.368,E2 -28947.368} C_VEL
LIN {X 0,Y 97.538,Z 712.723,A -85,B 0,C 180,E1 -28949.839,E2 -28949.839} C_VEL
LIN {X 0,Y 96.959,Z 712.457,A -85,B 0,C 180,E1 -28950.434,E2 -28950.434} C_VEL
LIN {X 0,Y 86.116,Z 708.69,A -85,B 0,C 180,E1 -28955.919,E2 -28955.919} C_VEL
LIN {X 0,Y 78.018,Z 704.37,A -85,B 0,C 180,E1 -28961.624,E2 -28961.624} C_VEL
LIN {X 0,Y 69.942,Z 697.898,A -85,B 0,C 180,E1 -28969.874,E2 -28969.874} C_VEL
LIN {X 0,Y 64.54,Z 690.977,A -85,B 0,C 180,E1 -28978.442,E2 -28978.442} C_VEL
LIN {X 0,Y 60.949,Z 682.514,A -85,B 0,C 180,E1 -28988.29,E2 -28988.29} C_VEL
LIN {X 0,Y 59.313,Z 672.662,A -85,B 0,C 180,E1 -28998.579,E2 -28998.579} C_VEL
LIN {X 0,Y 59.407,Z 662.614,A -85,B 0,C 180,E1 -29007.288,E2 -29007.288} C_VEL
LIN {X 0,Y 60.309,Z 652.585,A -85,B 0,C 180,E1 -29014.323,E2 -29014.323} C_VEL
LIN {X 0,Y 61.782,Z 641.083,A -85,B 0,C 180,E1 -29020.639,E2 -29020.639} C_VEL
LIN {X 0,Y 63.587,Z 628.156,A -85,B 0,C 180,E1 -29025.927,E2 -29025.927} C_VEL
LIN {X 0,Y 65.133,Z 615.085,A -85,B 0,C 180,E1 -29029.655,E2 -29029.655} C_VEL
LIN {X 0,Y 65.335,Z 613.431,A -85,B 0,C 180,E1 -29030.043,E2 -29030.043} C_VEL
LIN {X 0,Y 65.287,Z 609.62,A -85,B 0,C 180,E1 -29030.883,E2 -29030.883} C_VEL
LIN {X 0,Y 63.955,Z 604.004,A -85,B 0,C 180,E1 -29032.095,E2 -29032.095} C_VEL
LIN {X 0,Y 61.706,Z 598.613,A -85,B 0,C 180,E1 -29033.298,E2 -29033.298} C_VEL
LIN {X 0,Y 56.608,Z 587.755,A -85,B 0,C 180,E1 -29035.984,E2 -29035.984} C_VEL
LIN {X 0,Y 55.397,Z 583.971,A -85,B 0,C 180,E1 -29036.979,E2 -29036.979} C_VEL
LIN {X 0,Y 51.468,Z 569.964,A -85,B 0,C 180,E1 -29041.173,E2 -29041.173} C_VEL
LIN {X 0,Y 51.193,Z 569.012,A -85,B 0,C 180,E1 -29042.676,E2 -29042.676} C_VEL
LIN {X 0,Y 51.458,Z 568.878,A -85,B 0,C 180,E1 -29054.149,E2 -29054.149} C_VEL
LIN {X 0,Y 51.679,Z 568.85,A -85,B 0,C 180,E1 -29062.185,E2 -29062.185} C_VEL
LIN {X 0,Y 52.27,Z 568.778,A -85,B 0,C 180,E1 -29070.001,E2 -29070.001} C_VEL
LIN {X 0,Y 51.679,Z 568.855,A -85,B 0,C 180,E1 -29077.816,E2 -29077.816} C_VEL
LIN {X 0,Y 51.39,Z 568.891,A -85,B 0,C 180,E1 -29086.791,E2 -29086.791} C_VEL
LIN {X 0,Y 51.028,Z 568.941,A -85,B 0,C 180,E1 -29094.405,E2 -29094.405} C_VEL
LIN {X 0,Y 51.04,Z 568.936,A -85,B 0,C 180,E1 -29104.287,E2 -29104.287} C_VEL
LIN {X 0,Y 50.998,Z 568.935,A -85,B 0,C 180,E1 -29116.441,E2 -29116.441} C_VEL
LIN {X 0,Y 51.056,Z 568.93,A -85,B 0,C 180,E1 -29126.588,E2 -29126.588} C_VEL
LIN {X 0,Y 51.029,Z 568.934,A -85,B 0,C 180,E1 -29135.592,E2 -29135.592} C_VEL
LIN {X 0,Y 51.482,Z 568.877,A -85,B 0,C 180,E1 -29144.153,E2 -29144.153} C_VEL
LIN {X 0,Y 51.695,Z 568.848,A -85,B 0,C 180,E1 -29152.184,E2 -29152.184} C_VEL
LIN {X 0,Y 52.275,Z 568.776,A -85,B 0,C 180,E1 -29159.997,E2 -29159.997} C_VEL
LIN {X 0,Y 51.69,Z 568.85,A -85,B 0,C 180,E1 -29167.812,E2 -29167.812} C_VEL
LIN {X 0,Y 51.392,Z 568.887,A -85,B 0,C 180,E1 -29176.813,E2 -29176.813} C_VEL
LIN {X 0,Y 51.022,Z 568.938,A -85,B 0,C 180,E1 -29184.405,E2 -29184.405} C_VEL
LIN {X 0,Y 51.03,Z 568.933,A -85,B 0,C 180,E1 -29194.276,E2 -29194.276} C_VEL
LIN {X 0,Y 51.218,Z 569.011,A -85,B 0,C 180,E1 -29206.895,E2 -29206.895} C_VEL
LIN {X 0,Y 51.491,Z 569.903,A -85,B 0,C 180,E1 -29208.337,E2 -29208.337} C_VEL
LIN {X 0,Y 54.333,Z 578.604,A -85,B 0,C 180,E1 -29211.166,E2 -29211.166} C_VEL
LIN {X 0,Y 54.249,Z 623.331,A -85,B 0,C 180,E1 -29221.698,E2 -29221.698} C_VEL
LIN {X 0,Y 54.922,Z 638.026,A -85,B 0,C 180,E1 -29225.492,E2 -29225.492} C_VEL
LIN {X 0,Y 55.918,Z 652.195,A -85,B 0,C 180,E1 -29230.736,E2 -29230.736} C_VEL
LIN {X 0,Y 55.93,Z 659.776,A -85,B 0,C 180,E1 -29234.513,E2 -29234.513} C_VEL
LIN {X 0,Y 55.747,Z 668.636,A -85,B 0,C 180,E1 -29240.017,E2 -29240.017} C_VEL
LIN {X 0,Y 56.111,Z 679.395,A -85,B 0,C 180,E1 -29248.546,E2 -29248.546} C_VEL
LIN {X 0,Y 57.698,Z 688.144,A -85,B 0,C 180,E1 -29256.996,E2 -29256.996} C_VEL
LIN {X 0,Y 58.718,Z 691.523,A -85,B 0,C 180,E1 -29260.733,E2 -29260.733} C_VEL
LIN {X 0,Y 58.213,Z 696.58,A -85,B 0,C 180,E1 -29271.233,E2 -29271.233} C_VEL
LIN {X 0,Y 61.156,Z 702.032,A -85,B 0,C 180,E1 -29285.07,E2 -29285.07} C_VEL
LIN {X 0,Y 64.106,Z 704.251,A -85,B 0,C 180,E1 -29291.129,E2 -29291.129} C_VEL
LIN {X 0,Y 72.309,Z 707.713,A -85,B 0,C 180,E1 -29301.035,E2 -29301.035} C_VEL
LIN {X 0,Y 82.6,Z 709.977,A -85,B 0,C 180,E1 -29308.301,E2 -29308.301} C_VEL
LIN {X 0,Y 85.18,Z 710.154,A -85,B 0,C 180,E1 -29310.329,E2 -29310.329} C_VEL
LIN {X 0,Y 75.901,Z 705.729,A -85,B 0,C 180,E1 -29315.705,E2 -29315.705} C_VEL
LIN {X 0,Y 66.854,Z 699.354,A -85,B 0,C 180,E1 -29323.385,E2 -29323.385} C_VEL
LIN {X 0,Y 60.479,Z 692.676,A -85,B 0,C 180,E1 -29331.65,E2 -29331.65} C_VEL
LIN {X 0,Y 55.746,Z 684.592,A -85,B 0,C 180,E1 -29341.626,E2 -29341.626} C_VEL
LIN {X 0,Y 52.935,Z 674.299,A -85,B 0,C 180,E1 -29353.438,E2 -29353.438} C_VEL
LIN {X 0,Y 52.395,Z 663.936,A -85,B 0,C 180,E1 -29363.732,E2 -29363.732} C_VEL
LIN {X 0,Y 53.058,Z 653.839,A -85,B 0,C 180,E1 -29371.998,E2 -29371.998} C_VEL
LIN {X 0,Y 54.439,Z 642.417,A -85,B 0,C 180,E1 -29379.235,E2 -29379.235} C_VEL
LIN {X 0,Y 56.248,Z 629.456,A -85,B 0,C 180,E1 -29385.29,E2 -29385.29} C_VEL
LIN {X 0,Y 57.929,Z 616.204,A -85,B 0,C 180,E1 -29389.565,E2 -29389.565} C_VEL
LIN {X 0,Y 59.553,Z 599.062,A -85,B 0,C 180,E1 -29393.257,E2 -29393.257} C_VEL
LIN {X 0,Y 55.397,Z 583.971,A -85,B 0,C 180,E1 -29396.979,E2 -29396.979} C_VEL
LIN {X 0,Y 53.864,Z 581.642,A -85,B 0,C 180,E1 -29397.765,E2 -29397.765} C_VEL
LIN {X 0,Y 47.116,Z 577.311,A -85,B 0,C 180,E1 -29400.211,E2 -29400.211} C_VEL
LIN {X 0,Y 45.745,Z 575.3,A -85,B 0,C 180,E1 -29401.063,E2 -29401.063} C_VEL
LIN {X 0,Y 44.228,Z 570.54,A -85,B 0,C 180,E1 -29403.137,E2 -29403.137} C_VEL
LIN {X 0,Y 44.087,Z 569.84,A -85,B 0,C 180,E1 -29405.264,E2 -29405.264} C_VEL
LIN {X 0,Y 44.229,Z 569.778,A -85,B 0,C 180,E1 -29412.45,E2 -29412.45} C_VEL
LIN {X 0,Y 44.531,Z 569.742,A -85,B 0,C 180,E1 -29420.92,E2 -29420.92} C_VEL
LIN {X 0,Y 45.144,Z 569.665,A -85,B 0,C 180,E1 -29430.001,E2 -29430.001} C_VEL
LIN {X 0,Y 44.532,Z 569.741,A -85,B 0,C 180,E1 -29439.081,E2 -29439.081} C_VEL
LIN {X 0,Y 44.156,Z 569.787,A -85,B 0,C 180,E1 -29448.562,E2 -29448.562} C_VEL
LIN {X 0,Y 43.85,Z 569.825,A -85,B 0,C 180,E1 -29458.739,E2 -29458.739} C_VEL
LIN {X 0,Y 43.815,Z 569.836,A -85,B 0,C 180,E1 -29469.911,E2 -29469.911} C_VEL
LIN {X 0,Y 43.849,Z 569.826,A -85,B 0,C 180,E1 -29483.262,E2 -29483.262} C_VEL
LIN {X 0,Y 43.848,Z 569.83,A -85,B 0,C 180,E1 -29491.256,E2 -29491.256} C_VEL
LIN {X 0,Y 44.259,Z 569.774,A -85,B 0,C 180,E1 -29502.317,E2 -29502.317} C_VEL
LIN {X 0,Y 44.549,Z 569.738,A -85,B 0,C 180,E1 -29510.92,E2 -29510.92} C_VEL
LIN {X 0,Y 45.149,Z 569.663,A -85,B 0,C 180,E1 -29519.997,E2 -29519.997} C_VEL
LIN {X 0,Y 44.541,Z 569.739,A -85,B 0,C 180,E1 -29529.075,E2 -29529.075} C_VEL
LIN {X 0,Y 44.155,Z 569.787,A -85,B 0,C 180,E1 -29538.559,E2 -29538.559} C_VEL
LIN {X 0,Y 43.842,Z 569.828,A -85,B 0,C 180,E1 -29548.741,E2 -29548.741} C_VEL
LIN {X 0,Y 43.862,Z 569.834,A -85,B 0,C 180,E1 -29559.857,E2 -29559.857} C_VEL
LIN {X 0,Y 44.112,Z 570.081,A -85,B 0,C 180,E1 -29565.595,E2 -29565.595} C_VEL
LIN {X 0,Y 44.499,Z 571.334,A -85,B 0,C 180,E1 -29566.921,E2 -29566.921} C_VEL
LIN {X 0,Y 47.299,Z 579.501,A -85,B 0,C 180,E1 -29570.004,E2 -29570.004} C_VEL
LIN {X 0,Y 47.321,Z 627.47,A -85,B 0,C 180,E1 -29583.007,E2 -29583.007} C_VEL
LIN {X 0,Y 48.099,Z 640.845,A -85,B 0,C 180,E1 -29587.446,E2 -29587.446} C_VEL
LIN {X 0,Y 49.155,Z 653.82,A -85,B 0,C 180,E1 -29593.384,E2 -29593.384} C_VEL
LIN {X 0,Y 49.105,Z 663.791,A -85,B 0,C 180,E1 -29599.694,E2 -29599.694} C_VEL
LIN {X 0,Y 49.346,Z 673.819,A -85,B 0,C 180,E1 -29607.959,E2 -29607.959} C_VEL
LIN {X 0,Y 50.755,Z 682.526,A -85,B 0,C 180,E1 -29616.476,E2 -29616.476} C_VEL
LIN {X 0,Y 52.247,Z 687.518,A -85,B 0,C 180,E1 -29622.082,E2 -29622.082} C_VEL
LIN {X 0,Y 52.47,Z 689.64,A -85,B 0,C 180,E1 -29625.538,E2 -29625.538} C_VEL
LIN {X 0,Y 53.658,Z 696.225,A -85,B 0,C 180,E1 -29641.593,E2 -29641.593} C_VEL
LIN {X 0,Y 58.607,Z 700.864,A -85,B 0,C 180,E1 -29653.99,E2 -29653.99} C_VEL
LIN {X 0,Y 63.529,Z 703.399,A -85,B 0,C 180,E1 -29660.747,E2 -29660.747} C_VEL
LIN {X 0,Y 73.603,Z 706.629,A -85,B 0,C 180,E1 -29669.243,E2 -29669.243} C_VEL
LIN {X 0,Y 72.278,Z 705.676,A -85,B 0,C 180,E1 -29670.912,E2 -29670.912} C_VEL
LIN {X 0,Y 62.319,Z 698.929,A -85,B 0,C 180,E1 -29678.501,E2 -29678.501} C_VEL
LIN {X 0,Y 54.084,Z 690.409,A -85,B 0,C 180,E1 -29688.763,E2 -29688.763} C_VEL
LIN {X 0,Y 48.974,Z 681.481,A -85,B 0,C 180,E1 -29700.003,E2 -29700.003} C_VEL
LIN {X 0,Y 46.392,Z 672.555,A -85,B 0,C 180,E1 -29710.919,E2 -29710.919} C_VEL
LIN {X 0,Y 45.639,Z 662.79,A -85,B 0,C 180,E1 -29721.542,E2 -29721.542} C_VEL
LIN {X 0,Y 46.186,Z 652.388,A -85,B 0,C 180,E1 -29730.905,E2 -29730.905} C_VEL
LIN {X 0,Y 47.527,Z 640.693,A -85,B 0,C 180,E1 -29739.118,E2 -29739.118} C_VEL
LIN {X 0,Y 49.256,Z 628.191,A -85,B 0,C 180,E1 -29745.518,E2 -29745.518} C_VEL
LIN {X 0,Y 50.92,Z 615.316,A -85,B 0,C 180,E1 -29750.042,E2 -29750.042} C_VEL
LIN {X 0,Y 52.289,Z 599.27,A -85,B 0,C 180,E1 -29753.869,E2 -29753.869} C_VEL
LIN {X 0,Y 45.745,Z 575.3,A -85,B 0,C 180,E1 -29761.063,E2 -29761.063} C_VEL
LIN {X 0,Y 44.512,Z 572.943,A -85,B 0,C 180,E1 -29762.948,E2 -29762.948} C_VEL
LIN {X 0,Y 42.629,Z 571.187,A -85,B 0,C 180,E1 -29767.035,E2 -29767.035} C_VEL
LIN {X 0,Y 40.335,Z 570.373,A -85,B 0,C 180,E1 -29774.37,E2 -29774.37} C_VEL
LIN {X 0,Y 37.928,Z 570.563,A -85,B 0,C 180,E1 -29790.122,E2 -29790.122} C_VEL
LIN {X 0,Y 37.302,Z 570.64,A -85,B 0,C 180,E1 -29800.369,E2 -29800.369} C_VEL
LIN {X 0,Y 37.145,Z 570.65,A -85,B 0,C 180,E1 -29803.822,E2 -29803.822} C_VEL
LIN {X 0,Y 36.821,Z 570.707,A -85,B 0,C 180,E1 -29812.442,E2 -29812.442} C_VEL
LIN {X 0,Y 36.731,Z 570.714,A -85,B 0,C 180,E1 -29825.03,E2 -29825.03} C_VEL
LIN {X 0,Y 36.734,Z 570.717,A -85,B 0,C 180,E1 -29830.062,E2 -29830.062} C_VEL
LIN {X 0,Y 36.733,Z 570.722,A -85,B 0,C 180,E1 -29839.934,E2 -29839.934} C_VEL
LIN {X 0,Y 36.728,Z 570.711,A -85,B 0,C 180,E1 -29844.961,E2 -29844.961} C_VEL
LIN {X 0,Y 37.081,Z 570.668,A -85,B 0,C 180,E1 -29861.377,E2 -29861.377} C_VEL
LIN {X 0,Y 37.348,Z 570.638,A -85,B 0,C 180,E1 -29869.15,E2 -29869.15} C_VEL
LIN {X 0,Y 38.008,Z 570.552,A -85,B 0,C 180,E1 -29879.996,E2 -29879.996} C_VEL
LIN {X 0,Y 37.335,Z 570.638,A -85,B 0,C 180,E1 -29890.846,E2 -29890.846} C_VEL
LIN {X 0,Y 37.056,Z 570.671,A -85,B 0,C 180,E1 -29898.507,E2 -29898.507} C_VEL
LIN {X 0,Y 36.743,Z 570.71,A -85,B 0,C 180,E1 -29915.012,E2 -29915.012} C_VEL
LIN {X 0,Y 36.926,Z 570.918,A -85,B 0,C 180,E1 -29922.868,E2 -29922.868} C_VEL
LIN {X 0,Y 37.186,Z 571.707,A -85,B 0,C 180,E1 -29924.4,E2 -29924.4} C_VEL
LIN {X 0,Y 40.287,Z 581.086,A -85,B 0,C 180,E1 -29928.739,E2 -29928.739} C_VEL
LIN {X 0,Y 40.191,Z 626.971,A -85,B 0,C 180,E1 -29943.335,E2 -29943.335} C_VEL
LIN {X 0,Y 41.057,Z 640.509,A -85,B 0,C 180,E1 -29948.696,E2 -29948.696} C_VEL
LIN {X 0,Y 42.312,Z 653.27,A -85,B 0,C 180,E1 -29955.573,E2 -29955.573} C_VEL
LIN {X 0,Y 42.502,Z 662.97,A -85,B 0,C 180,E1 -29962.788,E2 -29962.788} C_VEL
LIN {X 0,Y 43.224,Z 673.029,A -85,B 0,C 180,E1 -29972.486,E2 -29972.486} C_VEL
LIN {X 0,Y 45.019,Z 680.726,A -85,B 0,C 180,E1 -29980.974,E2 -29980.974} C_VEL
LIN {X 0,Y 46.236,Z 684.183,A -85,B 0,C 180,E1 -29985.15,E2 -29985.15} C_VEL
LIN {X 0,Y 46.742,Z 685.807,A -85,B 0,C 180,E1 -29987.5,E2 -29987.5} C_VEL
LIN {X 0,Y 47.519,Z 691.244,A -85,B 0,C 180,E1 -30001.173,E2 -30001.173} C_VEL
LIN {X 0,Y 53.03,Z 697.006,A -85,B 0,C 180,E1 -30016.755,E2 -30016.755} C_VEL
LIN {X 0,Y 61.269,Z 701.199,A -85,B 0,C 180,E1 -30027.173,E2 -30027.173} C_VEL
LIN {X 0,Y 63.209,Z 701.813,A -85,B 0,C 180,E1 -30029.288,E2 -30029.288} C_VEL
LIN {X 0,Y 54.051,Z 694.572,A -85,B 0,C 180,E1 -30037.044,E2 -30037.044} C_VEL
LIN {X 0,Y 46.872,Z 686.313,A -85,B 0,C 180,E1 -30047.006,E2 -30047.006} C_VEL
LIN {X 0,Y 41.703,Z 676.34,A -85,B 0,C 180,E1 -30060.003,E2 -30060.003} C_VEL
LIN {X 0,Y 39.281,Z 665.171,A -85,B 0,C 180,E1 -30074.245,E2 -30074.245} C_VEL
LIN {X 0,Y 39.152,Z 654.312,A -85,B 0,C 180,E1 -30086.17,E2 -30086.17} C_VEL
LIN {X 0,Y 40.205,Z 642.593,A -85,B 0,C 180,E1 -30096.16,E2 -30096.16} C_VEL
LIN {X 0,Y 41.683,Z 631.219,A -85,B 0,C 180,E1 -30103.367,E2 -30103.367} C_VEL
LIN {X 0,Y 43.489,Z 617.738,A -85,B 0,C 180,E1 -30109.275,E2 -30109.275} C_VEL
LIN {X 0,Y 45.207,Z 600.817,A -85,B 0,C 180,E1 -30114.159,E2 -30114.159} C_VEL
LIN {X 0,Y 38.687,Z 576.202,A -85,B 0,C 180,E1 -30122.795,E2 -30122.795} C_VEL
LIN {X 0,Y 37.2,Z 571.567,A -85,B 0,C 180,E1 -30125.222,E2 -30125.222} C_VEL
LIN {X 0,Y 37.048,Z 570.817,A -85,B 0,C 180,E1 -30126.969,E2 -30126.969} C_VEL
LIN {X 0,Y 37.329,Z 570.644,A -85,B 0,C 180,E1 -30139.149,E2 -30139.149} C_VEL
LIN {X 0,Y 38.002,Z 570.554,A -85,B 0,C 180,E1 -30150.001,E2 -30150.001} C_VEL
LIN {X 0,Y 37.145,Z 570.65,A -85,B 0,C 180,E1 -30163.822,E2 -30163.822} C_VEL
LIN {X 0,Y 36.279,Z 570.771,A -85,B 0,C 180,E1 -30169.734,E2 -30169.734} C_VEL
LIN {X 0,Y 34.649,Z 570.974,A -85,B 0,C 180,E1 -30175.558,E2 -30175.558} C_VEL
LIN {X 0,Y 29.355,Z 571.479,A -85,B 0,C 180,E1 -30198.726,E2 -30198.726} C_VEL
LIN {X 0,Y 29.512,Z 571.483,A -85,B 0,C 180,E1 -30211.552,E2 -30211.552} C_VEL
LIN {X 0,Y 29.891,Z 571.448,A -85,B 0,C 180,E1 -30220.134,E2 -30220.134} C_VEL
LIN {X 0,Y 30.127,Z 571.428,A -85,B 0,C 180,E1 -30226.505,E2 -30226.505} C_VEL
LIN {X 0,Y 30.826,Z 571.358,A -85,B 0,C 180,E1 -30239.995,E2 -30239.995} C_VEL
LIN {X 0,Y 30.109,Z 571.43,A -85,B 0,C 180,E1 -30253.494,E2 -30253.494} C_VEL
LIN {X 0,Y 29.863,Z 571.45,A -85,B 0,C 180,E1 -30259.721,E2 -30259.721} C_VEL
LIN {X 0,Y 29.724,Z 571.525,A -85,B 0,C 180,E1 -30278.358,E2 -30278.358} C_VEL
LIN {X 0,Y 29.975,Z 572.473,A -85,B 0,C 180,E1 -30281.251,E2 -30281.251} C_VEL
LIN {X 0,Y 33.192,Z 581.653,A -85,B 0,C 180,E1 -30286.838,E2 -30286.838} C_VEL
LIN {X 0,Y 33.367,Z 630.502,A -85,B 0,C 180,E1 -30305.915,E2 -30305.915} C_VEL
LIN {X 0,Y 34.457,Z 643.747,A -85,B 0,C 180,E1 -30312.95,E2 -30312.95} C_VEL
LIN {X 0,Y 35.605,Z 653.388,A -85,B 0,C 180,E1 -30319.477,E2 -30319.477} C_VEL
LIN {X 0,Y 36.169,Z 662.483,A -85,B 0,C 180,E1 -30327.725,E2 -30327.725} C_VEL
LIN {X 0,Y 37.703,Z 672.891,A -85,B 0,C 180,E1 -30339.393,E2 -30339.393} C_VEL
LIN {X 0,Y 40.766,Z 681.529,A -85,B 0,C 180,E1 -30350.168,E2 -30350.168} C_VEL
LIN {X 0,Y 41.154,Z 683.095,A -85,B 0,C 180,E1 -30353.164,E2 -30353.164} C_VEL
LIN {X 0,Y 43.634,Z 689.201,A -85,B 0,C 180,E1 -30370.109,E2 -30370.109} C_VEL
LIN {X 0,Y 51.208,Z 695.032,A -85,B 0,C 180,E1 -30385.43,E2 -30385.43} C_VEL
LIN {X 0,Y 53.119,Z 695.983,A -85,B 0,C 180,E1 -30388.05,E2 -30388.05} C_VEL
LIN {X 0,Y 44.885,Z 688.11,A -85,B 0,C 180,E1 -30396.471,E2 -30396.471} C_VEL
LIN {X 0,Y 37.768,Z 678.121,A -85,B 0,C 180,E1 -30409.28,E2 -30409.28} C_VEL
LIN {X 0,Y 33.73,Z 667.165,A -85,B 0,C 180,E1 -30424.486,E2 -30424.486} C_VEL
LIN {X 0,Y 32.512,Z 656.328,A -85,B 0,C 180,E1 -30438.925,E2 -30438.925} C_VEL
LIN {X 0,Y 33.066,Z 643.652,A -85,B 0,C 180,E1 -30452.558,E2 -30452.558} C_VEL
LIN {X 0,Y 34.424,Z 632.175,A -85,B 0,C 180,E1 -30461.574,E2 -30461.574} C_VEL
LIN {X 0,Y 36.244,Z 618.737,A -85,B 0,C 180,E1 -30468.718,E2 -30468.718} C_VEL
LIN {X 0,Y 38.07,Z 601.093,A -85,B 0,C 180,E1 -30474.77,E2 -30474.77} C_VEL
LIN {X 0,Y 31.62,Z 577.065,A -85,B 0,C 180,E1 -30485.233,E2 -30485.233} C_VEL
LIN {X 0,Y 30.136,Z 572.299,A -85,B 0,C 180,E1 -30488.351,E2 -30488.351} C_VEL
LIN {X 0,Y 30.032,Z 571.491,A -85,B 0,C 180,E1 -30491.069,E2 -30491.069} C_VEL
LIN {X 0,Y 30.127,Z 571.425,A -85,B 0,C 180,E1 -30496.511,E2 -30496.511} C_VEL
LIN {X 0,Y 30.819,Z 571.359,A -85,B 0,C 180,E1 -30510.001,E2 -30510.001} C_VEL
LIN {X 0,Y 30.108,Z 571.429,A -85,B 0,C 180,E1 -30523.5,E2 -30523.5} C_VEL
LIN {X 0,Y 29.867,Z 571.448,A -85,B 0,C 180,E1 -30529.725,E2 -30529.725} C_VEL
LIN {X 0,Y 29.501,Z 571.483,A -85,B 0,C 180,E1 -30538.455,E2 -30538.455} C_VEL
LIN {X 0,Y 29.547,Z 571.478,A -85,B 0,C 180,E1 -30555.527,E2 -30555.527} C_VEL
LIN {X 0,Y 29.355,Z 571.479,A -85,B 0,C 180,E1 -30558.726,E2 -30558.726} C_VEL
LIN {X 0,Y 28.625,Z 571.566,A -85,B 0,C 180,E1 -30566.493,E2 -30566.493} C_VEL
LIN {X 0,Y 26.948,Z 571.721,A -85,B 0,C 180,E1 -30577.039,E2 -30577.039} C_VEL
LIN {X 0,Y 24.574,Z 571.836,A -85,B 0,C 180,E1 -30591.601,E2 -30591.601} C_VEL
LIN {X 0,Y 23.163,Z 571.86,A -85,B 0,C 180,E1 -30604.674,E2 -30604.674} C_VEL
LIN {X 0,Y 22.813,Z 571.878,A -85,B 0,C 180,E1 -30617.936,E2 -30617.936} C_VEL
LIN {X 0,Y 22.486,Z 572.14,A -85,B 0,C 180,E1 -30633.635,E2 -30633.635} C_VEL
LIN {X 0,Y 22.855,Z 573.392,A -85,B 0,C 180,E1 -30636.685,E2 -30636.685} C_VEL
LIN {X 0,Y 26.192,Z 582.865,A -85,B 0,C 180,E1 -30644.32,E2 -30644.32} C_VEL
LIN {X 0,Y 26.331,Z 630.263,A -85,B 0,C 180,E1 -30667.954,E2 -30667.954} C_VEL
LIN {X 0,Y 27.585,Z 642.606,A -85,B 0,C 180,E1 -30676.158,E2 -30676.158} C_VEL
LIN {X 0,Y 29.099,Z 652.569,A -85,B 0,C 180,E1 -30684.338,E2 -30684.338} C_VEL
LIN {X 0,Y 30.067,Z 660.926,A -85,B 0,C 180,E1 -30693.349,E2 -30693.349} C_VEL
LIN {X 0,Y 32.559,Z 671.773,A -85,B 0,C 180,E1 -30707.264,E2 -30707.264} C_VEL
LIN {X 0,Y 35.803,Z 678.899,A -85,B 0,C 180,E1 -30716.882,E2 -30716.882} C_VEL
LIN {X 0,Y 39.235,Z 685.427,A -85,B 0,C 180,E1 -30735.764,E2 -30735.764} C_VEL
LIN {X 0,Y 43.117,Z 688.716,A -85,B 0,C 180,E1 -30744.583,E2 -30744.583} C_VEL
LIN {X 0,Y 42.926,Z 688.278,A -85,B 0,C 180,E1 -30746.9,E2 -30746.9} C_VEL
LIN {X 0,Y 35.445,Z 679.618,A -85,B 0,C 180,E1 -30756.641,E2 -30756.641} C_VEL
LIN {X 0,Y 29.543,Z 669.197,A -85,B 0,C 180,E1 -30771.205,E2 -30771.205} C_VEL
LIN {X 0,Y 26.595,Z 658.509,A -85,B 0,C 180,E1 -30787.598,E2 -30787.598} C_VEL
LIN {X 0,Y 26.08,Z 646.923,A -85,B 0,C 180,E1 -30803.848,E2 -30803.848} C_VEL
LIN {X 0,Y 27.104,Z 634.048,A -85,B 0,C 180,E1 -30817.628,E2 -30817.628} C_VEL
LIN {X 0,Y 28.893,Z 620.087,A -85,B 0,C 180,E1 -30827.482,E2 -30827.482} C_VEL
LIN {X 0,Y 30.885,Z 602.333,A -85,B 0,C 180,E1 -30835.24,E2 -30835.24} C_VEL
LIN {X 0,Y 29.39,Z 596.254,A -85,B 0,C 180,E1 -30838.021,E2 -30838.021} C_VEL
LIN {X 0,Y 25.047,Z 579.436,A -85,B 0,C 180,E1 -30847.673,E2 -30847.673} C_VEL
LIN {X 0,Y 23.066,Z 572.707,A -85,B 0,C 180,E1 -30853.404,E2 -30853.404} C_VEL
LIN {X 0,Y 23.043,Z 571.947,A -85,B 0,C 180,E1 -30856.778,E2 -30856.778} C_VEL
LIN {X 0,Y 23.589,Z 571.853,A -85,B 0,C 180,E1 -30870.001,E2 -30870.001} C_VEL
LIN {X 0,Y 22.816,Z 571.877,A -85,B 0,C 180,E1 -30887.942,E2 -30887.942} C_VEL
LIN {X 0,Y 22.199,Z 571.897,A -85,B 0,C 180,E1 -30909.286,E2 -30909.286} C_VEL
LIN {X 0,Y 22.202,Z 571.897,A -85,B 0,C 180,E1 -30920.713,E2 -30920.713} C_VEL
LIN {X 0,Y 22.842,Z 571.876,A -85,B 0,C 180,E1 -30942.074,E2 -30942.074} C_VEL
LIN {X 0,Y 23.594,Z 571.853,A -85,B 0,C 180,E1 -30959.994,E2 -30959.994} C_VEL
LIN {X 0,Y 23.163,Z 571.86,A -85,B 0,C 180,E1 -30964.674,E2 -30964.674} C_VEL
LIN {X 0,Y 22.638,Z 572.408,A -85,B 0,C 180,E1 -30971.236,E2 -30971.236} C_VEL
LIN {X 0,Y 21.965,Z 574.313,A -85,B 0,C 180,E1 -30979.201,E2 -30979.201} C_VEL
LIN {X 0,Y 21.187,Z 577.858,A -85,B 0,C 180,E1 -30987.706,E2 -30987.706} C_VEL
LIN {X 0,Y 20.239,Z 583.194,A -85,B 0,C 180,E1 -30995.741,E2 -30995.741} C_VEL
LIN {X 0,Y 19.292,Z 589.415,A -85,B 0,C 180,E1 -31002.527,E2 -31002.527} C_VEL
LIN {X 0,Y 18.632,Z 598.041,A -85,B 0,C 180,E1 -31009.588,E2 -31009.588} C_VEL
LIN {X 0,Y 19.324,Z 629.33,A -85,B 0,C 180,E1 -31031.225,E2 -31031.225} C_VEL
LIN {X 0,Y 21.018,Z 642.253,A -85,B 0,C 180,E1 -31042.459,E2 -31042.459} C_VEL
LIN {X 0,Y 22.993,Z 651.863,A -85,B 0,C 180,E1 -31052.188,E2 -31052.188} C_VEL
LIN {X 0,Y 24.886,Z 661.001,A -85,B 0,C 180,E1 -31064.305,E2 -31064.305} C_VEL
LIN {X 0,Y 28.846,Z 671.452,A -85,B 0,C 180,E1 -31079.159,E2 -31079.159} C_VEL
LIN {X 0,Y 31.072,Z 675.34,A -85,B 0,C 180,E1 -31084.425,E2 -31084.425} C_VEL
LIN {X 0,Y 32.192,Z 677.612,A -85,B 0,C 180,E1 -31090.913,E2 -31090.913} C_VEL
LIN {X 0,Y 33.335,Z 679.27,A -85,B 0,C 180,E1 -31096.079,E2 -31096.079} C_VEL
LIN {X 0,Y 34.995,Z 681.073,A -85,B 0,C 180,E1 -31102.957,E2 -31102.957} C_VEL
LIN {X 0,Y 26.542,Z 669.571,A -85,B 0,C 180,E1 -31116.604,E2 -31116.604} C_VEL
LIN {X 0,Y 21.538,Z 657.974,A -85,B 0,C 180,E1 -31135.326,E2 -31135.326} C_VEL
LIN {X 0,Y 19.717,Z 646.312,A -85,B 0,C 180,E1 -31155.513,E2 -31155.513} C_VEL
LIN {X 0,Y 20.153,Z 633.891,A -85,B 0,C 180,E1 -31173.026,E2 -31173.026} C_VEL
LIN {X 0,Y 21.671,Z 620.675,A -85,B 0,C 180,E1 -31185.577,E2 -31185.577} C_VEL
LIN {X 0,Y 23.765,Z 602.398,A -85,B 0,C 180,E1 -31196.123,E2 -31196.123} C_VEL
LIN {X 0,Y 18.577,Z 581.954,A -85,B 0,C 180,E1 -31211.387,E2 -31211.387} C_VEL
LIN {X 0,Y 16.117,Z 572.919,A -85,B 0,C 180,E1 -31222.957,E2 -31222.957} C_VEL
LIN {X 0,Y 16.251,Z 572.068,A -85,B 0,C 180,E1 -31228.453,E2 -31228.453} C_VEL
LIN {X 0,Y 15.261,Z 571.991,A -85,B 0,C 180,E1 -31252.895,E2 -31252.895} C_VEL
LIN {X 0,Y 15.072,Z 571.991,A -85,B 0,C 180,E1 -31257.795,E2 -31257.795} C_VEL
LIN {X 0,Y 15.111,Z 571.991,A -85,B 0,C 180,E1 -31292.274,E2 -31292.274} C_VEL
LIN {X 0,Y 15.29,Z 571.991,A -85,B 0,C 180,E1 -31296.828,E2 -31296.828} C_VEL
LIN {X 0,Y 16.254,Z 571.991,A -85,B 0,C 180,E1 -31320.083,E2 -31320.083} C_VEL
LIN {X 0,Y 15.525,Z 572.077,A -85,B 0,C 180,E1 -31339.748,E2 -31339.748} C_VEL
LIN {X 0,Y 15.42,Z 572.869,A -85,B 0,C 180,E1 -31344.974,E2 -31344.974} C_VEL
LIN {X 0,Y 18.107,Z 580.431,A -85,B 0,C 180,E1 -31356.642,E2 -31356.642} C_VEL
LIN {X 0,Y 19.318,Z 584.739,A -85,B 0,C 180,E1 -31360.889,E2 -31360.889} C_VEL
LIN {X 0,Y 18.632,Z 598.041,A -85,B 0,C 180,E1 -31369.588,E2 -31369.588} C_VEL
LIN {X 0,Y 17.951,Z 603.782,A -85,B 0,C 180,E1 -31373.306,E2 -31373.306} C_VEL
LIN {X 0,Y 12.666,Z 622.345,A -85,B 0,C 180,E1 -31390.763,E2 -31390.763} C_VEL
LIN {X 0,Y 12.469,Z 628.021,A -85,B 0,C 180,E1 -31398.285,E2 -31398.285} C_VEL
LIN {X 0,Y 14.712,Z 640.779,A -85,B 0,C 180,E1 -31413.421,E2 -31413.421} C_VEL
LIN {X 0,Y 17.486,Z 650.359,A -85,B 0,C 180,E1 -31424.546,E2 -31424.546} C_VEL
LIN {X 0,Y 20.027,Z 658.306,A -85,B 0,C 180,E1 -31436.016,E2 -31436.016} C_VEL
LIN {X 0,Y 25.316,Z 669.002,A -85,B 0,C 180,E1 -31451.246,E2 -31451.246} C_VEL
LIN {X 0,Y 26.532,Z 670.857,A -85,B 0,C 180,E1 -31453.498,E2 -31453.498} C_VEL
LIN {X 0,Y 27.327,Z 672.132,A -85,B 0,C 180,E1 -31457.546,E2 -31457.546} C_VEL
LIN {X 0,Y 19.888,Z 661.018,A -85,B 0,C 180,E1 -31470.938,E2 -31470.938} C_VEL
LIN {X 0,Y 15.469,Z 650.425,A -85,B 0,C 180,E1 -31489.653,E2 -31489.653} C_VEL
LIN {X 0,Y 13.551,Z 638.855,A -85,B 0,C 180,E1 -31513.507,E2 -31513.507} C_VEL
LIN {X 0,Y 13.898,Z 626.794,A -85,B 0,C 180,E1 -31534.685,E2 -31534.685} C_VEL
LIN {X 0,Y 15.33,Z 614.38,A -85,B 0,C 180,E1 -31548.297,E2 -31548.297} C_VEL
LIN {X 0,Y 16.568,Z 603.05,A -85,B 0,C 180,E1 -31557.241,E2 -31557.241} C_VEL
LIN {X 0,Y 12.06,Z 583.991,A -85,B 0,C 180,E1 -31579.51,E2 -31579.51} C_VEL
LIN {X 0,Y 10.543,Z 576.908,A -85,B 0,C 180,E1 -31593.757,E2 -31593.757} C_VEL
LIN {X 0,Y 8.653,Z 574.76,A -85,B 0,C 180,E1 -31610.635,E2 -31610.635} C_VEL
LIN {X 0,Y 7.826,Z 573.011,A -85,B 0,C 180,E1 -31653.911,E2 -31653.911} C_VEL
LIN {X 0,Y 9.179,Z 574.169,A -85,B 0,C 180,E1 -31682.232,E2 -31682.232} C_VEL
LIN {X 0,Y 9.983,Z 576.78,A -85,B 0,C 180,E1 -31692.481,E2 -31692.481} C_VEL
LIN {X 0,Y 11.995,Z 583.626,A -85,B 0,C 180,E1 -31709.637,E2 -31709.637} C_VEL
LIN {X 0,Y 12.486,Z 585.857,A -85,B 0,C 180,E1 -31713.258,E2 -31713.258} C_VEL
LIN {X 0,Y 12.469,Z 628.021,A -85,B 0,C 180,E1 -31758.285,E2 -31758.285} C_VEL
LIN {X 0,Y 12.284,Z 631.787,A -85,B 0,C 180,E1 -31764.328,E2 -31764.328} C_VEL
LIN {X 0,Y 11.176,Z 637.586,A -85,B 0,C 180,E1 -31780.453,E2 -31780.453} C_VEL
LIN {X 0,Y 11.356,Z 643.282,A -85,B 0,C 180,E1 -31798.944,E2 -31798.944} C_VEL
LIN {X 0,Y 12.576,Z 646.883,A -85,B 0,C 180,E1 -31804.808,E2 -31804.808} C_VEL
LIN {X 0,Y 15.261,Z 653.003,A -85,B 0,C 180,E1 -31810.894,E2 -31810.894} C_VEL
LIN {X 0,Y 15.371,Z 653.636,A -85,B 0,C 180,E1 -31816.789,E2 -31816.789} C_VEL
LIN {X 0,Y 10.298,Z 642.593,A -85,B 0,C 180,E1 -31834.885,E2 -31834.885} C_VEL
LIN {X 0,Y 7.565,Z 629.294,A -85,B 0,C 180,E1 -31869.339,E2 -31869.339} C_VEL
LIN {X 0,Y 8.113,Z 615.815,A -85,B 0,C 180,E1 -31900.939,E2 -31900.939} C_VEL
LIN {X 0,Y 9.273,Z 603.257,A -85,B 0,C 180,E1 -31919.822,E2 -31919.822} C_VEL
LIN {X 0,Y 6.214,Z 585.425,A -85,B 0,C 180,E1 -31965.156,E2 -31965.156} C_VEL
LIN {X 0,Y 6.131,Z 581.572,A -85,B 0,C 180,E1 -31982.001,E2 -31982.001} C_VEL
LIN {X 0,Y 5.947,Z 580.45,A -85,B 0,C 180,E1 -32009.585,E2 -32009.585} C_VEL
LIN {X 0,Y 6.102,Z 580.222,A -85,B 0,C 180,E1 -32016.122,E2 -32016.122} C_VEL
LIN {X 0,Y 6.399,Z 586.818,A -85,B 0,C 180,E1 -32049.418,E2 -32049.418} C_VEL
LIN {X 0,Y 6.239,Z 626.647,A -85,B 0,C 180,E1 -32140.372,E2 -32140.372} C_VEL
LIN {X 0,Y 9.719,Z 639.443,A -85,B 0,C 180,E1 -32157.859,E2 -32157.859} C_VEL
LIN {X 0,Y 12.576,Z 646.883,A -85,B 0,C 180,E1 -32164.808,E2 -32164.808} C_VEL
LIN {X 0,Y 12.576,Z 646.883,A -85,B 0,C 180,E1 -32164.808,E2 -32164.808}

QRS_NEXT_CUT()

QRS_NEXT()
QRS_HOME()

END
